KUKA KRL program: EPS_2_25252_SD6A_A_20250912064012.src

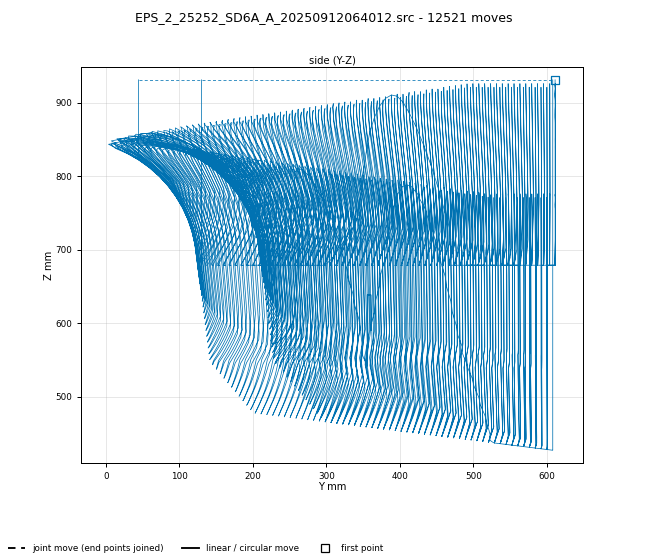
[picture p0: tool path of EPS_2_25252_SD6A_A_20250912064012.src, 12521 of 12523 moves have a stored position in this frame; points joined in program order, loops and branches not executed]
&ACCESS RVP
&REL 4
&COMMENT QRS 19112012
&PARAM EDITMASK = *
DEF PART()
EXT BAS (BAS_COMMAND :IN,REAL :IN )
INT I
BAS (#INITMOV,0 )

;KUKA QRS Post kuka4.cps  Date:22-06-2017 !

File_ID=2842

QRS_PRE_INIT()

;Init var - Until changes are made in qrs_pre_init
Outlet_Square_prg=0
Inlet_1_Square_prg=0
Inlet_2_Square_prg=0
Inlet_3_Square_prg=0
Inlet_4_Square_prg=0
Inlet_5_Square_prg=0

Outlet_1={X 0.000, Y 495.550, Z 738.000, B 0.000, E1 0.000 }
Inlet_1={X 0.000, Y 522.150, Z 645.500, B 0.000, E1 160.000 }
Outlet_1_type=366
Inlet_1_type=201
;QRS#1=Sidecore dimensions
;QRS#2=375-15" PVC SDR 35
;QRS#3=200-8" PVC SDR 35
;QRS#4=
;QRS#5=
;QRS#6=
;QRS#7=
;QRS#8=
;QRS#9=20Y PSX
;QRS#10=12-08 PSX
;QRS#11=
;QRS#12=
;QRS#13=
;QRS#14=
;QRS#15=
;QRS#16=1220x127x1219 4'
;QRS#17=EPS Height
;QRS#18=921
;QRS#19=*
;QRS#20= UPDATED VERSION 22-06-2017
;QRS#21=*
Outlet_Square=0250
Inlet_1_Square=0100
Inlet_2_Square=0
Inlet_3_Square=0
Inlet_4_Square=0
Inlet_5_Square=0
Mill_Square=1
Outlet_Square_Prg=252
Inlet_1_Square_prg=204

QRS_INIT()

$ADVANCE=5

; T1
PTP {E1 177.349,E2 177.349}
PTP {X 0,Y 611.1,A -85,B 0,C 180,E1 177.349,E2 177.349,E3 0,E4 0,E5 0,E6 0}
QRS_SPEED_INIT()
LIN {X 0,Y 611.1,Z 931,A -85,B 0,C 180,E1 177.349,E2 177.349,E3 0,E4 0,E5 0,E6 0} C_VEL
LIN {X 0,Y 611.1,Z 680.81,A -85,B 0,C 180,E1 177.349,E2 177.349} C_VEL
LIN {X 0,Y 611.172,Z 678.81,A -85,B 0,C 180,E1 177.537,E2 177.537} C_VEL
LIN {X 0,Y 611.853,Z 678.81,A -85,B 0,C 180,E1 178.833,E2 178.833} C_VEL
LIN {X 0,Y 611.873,Z 678.81,A -85,B 0,C 180,E1 185.845,E2 185.845} C_VEL
LIN {X 0,Y 611.832,Z 678.81,A -85,B 0,C 180,E1 192.946,E2 192.946} C_VEL
LIN {X 0,Y 611.828,Z 678.81,A -85,B 0,C 180,E1 200.258,E2 200.258} C_VEL
LIN {X 0,Y 611.823,Z 678.81,A -85,B 0,C 180,E1 207.934,E2 207.934} C_VEL
LIN {X 0,Y 610.481,Z 678.81,A -85,B 0,C 180,E1 210.684,E2 210.684} C_VEL
LIN {X 0,Y 611.798,Z 678.81,A -85,B 0,C 180,E1 216.206,E2 216.206} C_VEL
LIN {X 0,Y 611.214,Z 678.81,A -85,B 0,C 180,E1 217.333,E2 217.333} C_VEL
LIN {X 0,Y 610.734,Z 678.81,A -85,B 0,C 180,E1 222.325,E2 222.325} C_VEL
LIN {X 0,Y 611.755,Z 678.81,A -85,B 0,C 180,E1 224.525,E2 224.525} C_VEL
LIN {X 0,Y 611.734,Z 678.81,A -85,B 0,C 180,E1 232.604,E2 232.604} C_VEL
LIN {X 0,Y 611.207,Z 678.81,A -85,B 0,C 180,E1 233.754,E2 233.754} C_VEL
LIN {X 0,Y 611.701,Z 678.81,A -85,B 0,C 180,E1 241.161,E2 241.161} C_VEL
LIN {X 0,Y 611.507,Z 678.81,A -85,B 0,C 180,E1 242.05,E2 242.05} C_VEL
LIN {X 0,Y 611.773,Z 678.81,A -85,B 0,C 180,E1 248.631,E2 248.631} C_VEL
LIN {X 0,Y 610.949,Z 678.81,A -85,B 0,C 180,E1 248.984,E2 248.984} C_VEL
LIN {X 0,Y 610.788,Z 678.81,A -85,B 0,C 180,E1 249.001,E2 249.001} C_VEL
LIN {X 0,Y 611.596,Z 716.961,A -85,B 0,C 180,E1 249.507,E2 249.507} C_VEL
LIN {X 0,Y 611.806,Z 744.067,A -85,B 0,C 180,E1 249.858,E2 249.858} C_VEL
LIN {X 0,Y 611.827,Z 753.232,A -85,B 0,C 180,E1 250.014,E2 250.014} C_VEL
LIN {X 0,Y 611.806,Z 762.284,A -85,B 0,C 180,E1 250.207,E2 250.207} C_VEL
LIN {X 0,Y 611.661,Z 771.239,A -85,B 0,C 180,E1 250.435,E2 250.435} C_VEL
LIN {X 0,Y 611.79,Z 780.1,A -85,B 0,C 180,E1 250.71,E2 250.71} C_VEL
LIN {X 0,Y 611.791,Z 787.863,A -85,B 0,C 180,E1 250.98,E2 250.98} C_VEL
LIN {X 0,Y 611.787,Z 797.495,A -85,B 0,C 180,E1 251.365,E2 251.365} C_VEL
LIN {X 0,Y 611.804,Z 805.998,A -85,B 0,C 180,E1 251.75,E2 251.75} C_VEL
LIN {X 0,Y 611.73,Z 815.053,A -85,B 0,C 180,E1 252.208,E2 252.208} C_VEL
LIN {X 0,Y 611.709,Z 824.508,A -85,B 0,C 180,E1 252.747,E2 252.747} C_VEL
LIN {X 0,Y 611.546,Z 832.95,A -85,B 0,C 180,E1 253.278,E2 253.278} C_VEL
LIN {X 0,Y 611.448,Z 839.372,A -85,B 0,C 180,E1 253.718,E2 253.718} C_VEL
LIN {X 0,Y 611.513,Z 846.795,A -85,B 0,C 180,E1 254.279,E2 254.279} C_VEL
LIN {X 0,Y 611.729,Z 854.696,A -85,B 0,C 180,E1 254.937,E2 254.937} C_VEL
LIN {X 0,Y 611.827,Z 861.197,A -85,B 0,C 180,E1 255.523,E2 255.523} C_VEL
LIN {X 0,Y 611.641,Z 868.111,A -85,B 0,C 180,E1 256.198,E2 256.198} C_VEL
LIN {X 0,Y 611.381,Z 874.097,A -85,B 0,C 180,E1 256.831,E2 256.831} C_VEL
LIN {X 0,Y 611.254,Z 879.807,A -85,B 0,C 180,E1 257.49,E2 257.49} C_VEL
LIN {X 0,Y 611.36,Z 885.701,A -85,B 0,C 180,E1 258.239,E2 258.239} C_VEL
LIN {X 0,Y 611.556,Z 890.069,A -85,B 0,C 180,E1 258.838,E2 258.838} C_VEL
LIN {X 0,Y 611.862,Z 895.943,A -85,B 0,C 180,E1 259.735,E2 259.735} C_VEL
LIN {X 0,Y 611.484,Z 901.185,A -85,B 0,C 180,E1 260.617,E2 260.617} C_VEL
LIN {X 0,Y 611.211,Z 904.398,A -85,B 0,C 180,E1 261.204,E2 261.204} C_VEL
LIN {X 0,Y 611.059,Z 908.684,A -85,B 0,C 180,E1 262.088,E2 262.088} C_VEL
LIN {X 0,Y 611.226,Z 912.436,A -85,B 0,C 180,E1 262.974,E2 262.974} C_VEL
LIN {X 0,Y 611.629,Z 915.681,A -85,B 0,C 180,E1 263.86,E2 263.86} C_VEL
LIN {X 0,Y 611.768,Z 916.615,A -85,B 0,C 180,E1 264.154,E2 264.154} C_VEL
LIN {X 0,Y 611.736,Z 918.452,A -85,B 0,C 180,E1 264.74,E2 264.74} C_VEL
LIN {X 0,Y 611.169,Z 921.43,A -85,B 0,C 180,E1 265.908,E2 265.908} C_VEL
LIN {X 0,Y 610.976,Z 922.681,A -85,B 0,C 180,E1 266.492,E2 266.492} C_VEL
LIN {X 0,Y 611.094,Z 924.535,A -85,B 0,C 180,E1 267.712,E2 267.712} C_VEL
LIN {X 0,Y 611.599,Z 925.552,A -85,B 0,C 180,E1 268.833,E2 268.833} C_VEL
LIN {X 0,Y 611.822,Z 925.786,A -85,B 0,C 180,E1 269.3,E2 269.3} C_VEL
LIN {X 0,Y 611.469,Z 925.916,A -85,B 0,C 180,E1 270.234,E2 270.234} C_VEL
LIN {X 0,Y 611.076,Z 925.575,A -85,B 0,C 180,E1 271.168,E2 271.168} C_VEL
LIN {X 0,Y 611.003,Z 924.587,A -85,B 0,C 180,E1 272.246,E2 272.246} C_VEL
LIN {X 0,Y 611.445,Z 922.667,A -85,B 0,C 180,E1 273.505,E2 273.505} C_VEL
LIN {X 0,Y 611.74,Z 921.409,A -85,B 0,C 180,E1 274.088,E2 274.088} C_VEL
LIN {X 0,Y 611.75,Z 920.023,A -85,B 0,C 180,E1 274.674,E2 274.674} C_VEL
LIN {X 0,Y 611.456,Z 918.462,A -85,B 0,C 180,E1 275.262,E2 275.262} C_VEL
LIN {X 0,Y 611.035,Z 915.69,A -85,B 0,C 180,E1 276.146,E2 276.146} C_VEL
LIN {X 0,Y 610.903,Z 912.436,A -85,B 0,C 180,E1 277.03,E2 277.03} C_VEL
LIN {X 0,Y 611.131,Z 908.684,A -85,B 0,C 180,E1 277.911,E2 277.911} C_VEL
LIN {X 0,Y 611.584,Z 904.398,A -85,B 0,C 180,E1 278.79,E2 278.79} C_VEL
LIN {X 0,Y 611.866,Z 901.185,A -85,B 0,C 180,E1 279.377,E2 279.377} C_VEL
LIN {X 0,Y 611.515,Z 895.944,A -85,B 0,C 180,E1 280.271,E2 280.271} C_VEL
LIN {X 0,Y 611.151,Z 888.996,A -85,B 0,C 180,E1 281.318,E2 281.318} C_VEL
LIN {X 0,Y 611.162,Z 883.427,A -85,B 0,C 180,E1 282.063,E2 282.063} C_VEL
LIN {X 0,Y 611.413,Z 877.293,A -85,B 0,C 180,E1 282.806,E2 282.806} C_VEL
LIN {X 0,Y 611.786,Z 869.803,A -85,B 0,C 180,E1 283.623,E2 283.623} C_VEL
LIN {X 0,Y 611.787,Z 863.856,A -85,B 0,C 180,E1 284.223,E2 284.223} C_VEL
LIN {X 0,Y 611.564,Z 856.74,A -85,B 0,C 180,E1 284.888,E2 284.888} C_VEL
LIN {X 0,Y 611.414,Z 850.125,A -85,B 0,C 180,E1 285.456,E2 285.456} C_VEL
LIN {X 0,Y 611.435,Z 843.15,A -85,B 0,C 180,E1 286.003,E2 286.003} C_VEL
LIN {X 0,Y 611.594,Z 835.525,A -85,B 0,C 180,E1 286.548,E2 286.548} C_VEL
LIN {X 0,Y 611.771,Z 827.341,A -85,B 0,C 180,E1 287.078,E2 287.078} C_VEL
LIN {X 0,Y 611.809,Z 819.307,A -85,B 0,C 180,E1 287.555,E2 287.555} C_VEL
LIN {X 0,Y 611.791,Z 810.646,A -85,B 0,C 180,E1 288.02,E2 288.02} C_VEL
LIN {X 0,Y 611.702,Z 802.729,A -85,B 0,C 180,E1 288.407,E2 288.407} C_VEL
LIN {X 0,Y 611.705,Z 793.825,A -85,B 0,C 180,E1 288.791,E2 288.791} C_VEL
LIN {X 0,Y 611.795,Z 783.539,A -85,B 0,C 180,E1 289.174,E2 289.174} C_VEL
LIN {X 0,Y 611.762,Z 773.929,A -85,B 0,C 180,E1 289.485,E2 289.485} C_VEL
LIN {X 0,Y 611.767,Z 767.133,A -85,B 0,C 180,E1 289.678,E2 289.678} C_VEL
LIN {X 0,Y 611.841,Z 755.254,A -85,B 0,C 180,E1 289.947,E2 289.947} C_VEL
LIN {X 0,Y 611.828,Z 745.402,A -85,B 0,C 180,E1 290.122,E2 290.122} C_VEL
LIN {X 0,Y 611.684,Z 723.448,A -85,B 0,C 180,E1 290.41,E2 290.41} C_VEL
LIN {X 0,Y 610.946,Z 685.949,A -85,B 0,C 180,E1 290.897,E2 290.897} C_VEL
LIN {X 0,Y 610.763,Z 678.81,A -85,B 0,C 180,E1 290.996,E2 290.996} C_VEL
LIN {X 0,Y 611.68,Z 678.81,A -85,B 0,C 180,E1 291.148,E2 291.148} C_VEL
LIN {X 0,Y 611.713,Z 678.81,A -85,B 0,C 180,E1 291.751,E2 291.751} C_VEL
LIN {X 0,Y 611.826,Z 678.81,A -85,B 0,C 180,E1 300.61,E2 300.61} C_VEL
LIN {X 0,Y 610.649,Z 678.81,A -85,B 0,C 180,E1 307.263,E2 307.263} C_VEL
LIN {X 0,Y 611.78,Z 678.81,A -85,B 0,C 180,E1 309.156,E2 309.156} C_VEL
LIN {X 0,Y 610.375,Z 678.81,A -85,B 0,C 180,E1 312.355,E2 312.355} C_VEL
LIN {X 0,Y 610.685,Z 678.81,A -85,B 0,C 180,E1 315.577,E2 315.577} C_VEL
LIN {X 0,Y 611.769,Z 678.81,A -85,B 0,C 180,E1 317.764,E2 317.764} C_VEL
LIN {X 0,Y 610.272,Z 678.81,A -85,B 0,C 180,E1 323.689,E2 323.689} C_VEL
LIN {X 0,Y 611.793,Z 678.81,A -85,B 0,C 180,E1 326.636,E2 326.636} C_VEL
LIN {X 0,Y 611.803,Z 678.81,A -85,B 0,C 180,E1 334.676,E2 334.676} C_VEL
LIN {X 0,Y 611.537,Z 678.81,A -85,B 0,C 180,E1 343.281,E2 343.281} C_VEL
LIN {X 0,Y 611.296,Z 678.81,A -85,B 0,C 180,E1 344.633,E2 344.633} C_VEL
LIN {X 0,Y 611.872,Z 678.81,A -85,B 0,C 180,E1 351.804,E2 351.804} C_VEL
LIN {X 0,Y 611.852,Z 678.81,A -85,B 0,C 180,E1 358.833,E2 358.833} C_VEL
LIN {X 0,Y 611.874,Z 678.81,A -85,B 0,C 180,E1 368.196,E2 368.196} C_VEL
LIN {X 0,Y 611.806,Z 678.81,A -85,B 0,C 180,E1 375.354,E2 375.354} C_VEL
LIN {X 0,Y 611.825,Z 678.81,A -85,B 0,C 180,E1 382.767,E2 382.767} C_VEL
LIN {X 0,Y 611.831,Z 678.81,A -85,B 0,C 180,E1 390.609,E2 390.609} C_VEL
LIN {X 0,Y 611.757,Z 678.81,A -85,B 0,C 180,E1 399.158,E2 399.158} C_VEL
LIN {X 0,Y 610.337,Z 678.81,A -85,B 0,C 180,E1 402.359,E2 402.359} C_VEL
LIN {X 0,Y 610.636,Z 678.81,A -85,B 0,C 180,E1 405.582,E2 405.582} C_VEL
LIN {X 0,Y 611.712,Z 678.81,A -85,B 0,C 180,E1 407.759,E2 407.759} C_VEL
LIN {X 0,Y 610.218,Z 678.81,A -85,B 0,C 180,E1 413.686,E2 413.686} C_VEL
LIN {X 0,Y 611.725,Z 678.81,A -85,B 0,C 180,E1 416.637,E2 416.637} C_VEL
LIN {X 0,Y 611.755,Z 678.81,A -85,B 0,C 180,E1 424.674,E2 424.674} C_VEL
LIN {X 0,Y 611.523,Z 678.81,A -85,B 0,C 180,E1 433.285,E2 433.285} C_VEL
LIN {X 0,Y 611.29,Z 678.81,A -85,B 0,C 180,E1 434.632,E2 434.632} C_VEL
LIN {X 0,Y 611.873,Z 678.81,A -85,B 0,C 180,E1 441.804,E2 441.804} C_VEL
LIN {X 0,Y 611.873,Z 678.81,A -85,B 0,C 180,E1 448.833,E2 448.833} C_VEL
LIN {X 0,Y 611.836,Z 678.81,A -85,B 0,C 180,E1 457.976,E2 457.976} C_VEL
LIN {X 0,Y 611.68,Z 678.812,A -85,B 0,C 180,E1 458.051,E2 458.051} C_VEL
LIN {X 0,Y 611.823,Z 687.514,A -85,B 0,C 180,E1 458.307,E2 458.307} C_VEL
LIN {X 0,Y 611.725,Z 694.867,A -85,B 0,C 180,E1 458.567,E2 458.567} C_VEL
LIN {X 0,Y 611.706,Z 703.414,A -85,B 0,C 180,E1 458.936,E2 458.936} C_VEL
LIN {X 0,Y 611.787,Z 710.617,A -85,B 0,C 180,E1 459.304,E2 459.304} C_VEL
LIN {X 0,Y 611.823,Z 718.098,A -85,B 0,C 180,E1 459.747,E2 459.747} C_VEL
LIN {X 0,Y 611.74,Z 724.654,A -85,B 0,C 180,E1 460.193,E2 460.193} C_VEL
LIN {X 0,Y 611.547,Z 731.453,A -85,B 0,C 180,E1 460.716,E2 460.716} C_VEL
LIN {X 0,Y 611.554,Z 738.108,A -85,B 0,C 180,E1 461.31,E2 461.31} C_VEL
LIN {X 0,Y 611.754,Z 743.901,A -85,B 0,C 180,E1 461.902,E2 461.902} C_VEL
LIN {X 0,Y 611.846,Z 749.025,A -85,B 0,C 180,E1 462.498,E2 462.498} C_VEL
LIN {X 0,Y 611.57,Z 754.062,A -85,B 0,C 180,E1 463.155,E2 463.155} C_VEL
LIN {X 0,Y 611.352,Z 758.117,A -85,B 0,C 180,E1 463.768,E2 463.768} C_VEL
LIN {X 0,Y 611.348,Z 761.59,A -85,B 0,C 180,E1 464.365,E2 464.365} C_VEL
LIN {X 0,Y 611.521,Z 764.619,A -85,B 0,C 180,E1 464.961,E2 464.961} C_VEL
LIN {X 0,Y 611.856,Z 767.987,A -85,B 0,C 180,E1 465.746,E2 465.746} C_VEL
LIN {X 0,Y 611.76,Z 769.47,A -85,B 0,C 180,E1 466.142,E2 466.142} C_VEL
LIN {X 0,Y 611.48,Z 771.28,A -85,B 0,C 180,E1 466.702,E2 466.702} C_VEL
LIN {X 0,Y 611.285,Z 772.515,A -85,B 0,C 180,E1 467.157,E2 467.157} C_VEL
LIN {X 0,Y 611.186,Z 773.958,A -85,B 0,C 180,E1 467.808,E2 467.808} C_VEL
LIN {X 0,Y 611.315,Z 774.93,A -85,B 0,C 180,E1 468.419,E2 468.419} C_VEL
LIN {X 0,Y 611.592,Z 775.562,A -85,B 0,C 180,E1 469.026,E2 469.026} C_VEL
LIN {X 0,Y 611.86,Z 775.874,A -85,B 0,C 180,E1 469.636,E2 469.636} C_VEL
LIN {X 0,Y 611.627,Z 775.89,A -85,B 0,C 180,E1 470.265,E2 470.265} C_VEL
LIN {X 0,Y 611.328,Z 775.619,A -85,B 0,C 180,E1 470.822,E2 470.822} C_VEL
LIN {X 0,Y 611.148,Z 775.071,A -85,B 0,C 180,E1 471.378,E2 471.378} C_VEL
LIN {X 0,Y 611.15,Z 773.993,A -85,B 0,C 180,E1 472.083,E2 472.083} C_VEL
LIN {X 0,Y 611.421,Z 772.429,A -85,B 0,C 180,E1 472.783,E2 472.783} C_VEL
LIN {X 0,Y 611.84,Z 770.085,A -85,B 0,C 180,E1 473.578,E2 473.578} C_VEL
LIN {X 0,Y 611.755,Z 768.443,A -85,B 0,C 180,E1 474.044,E2 474.044} C_VEL
LIN {X 0,Y 611.36,Z 764.799,A -85,B 0,C 180,E1 474.914,E2 474.914} C_VEL
LIN {X 0,Y 611.234,Z 761.497,A -85,B 0,C 180,E1 475.563,E2 475.563} C_VEL
LIN {X 0,Y 611.357,Z 757.756,A -85,B 0,C 180,E1 476.201,E2 476.201} C_VEL
LIN {X 0,Y 611.664,Z 753.487,A -85,B 0,C 180,E1 476.834,E2 476.834} C_VEL
LIN {X 0,Y 611.854,Z 750.246,A -85,B 0,C 180,E1 477.263,E2 477.263} C_VEL
LIN {X 0,Y 611.7,Z 744.512,A -85,B 0,C 180,E1 477.94,E2 477.94} C_VEL
LIN {X 0,Y 611.466,Z 738.388,A -85,B 0,C 180,E1 478.575,E2 478.575} C_VEL
LIN {X 0,Y 611.482,Z 732.628,A -85,B 0,C 180,E1 479.094,E2 479.094} C_VEL
LIN {X 0,Y 611.679,Z 725.889,A -85,B 0,C 180,E1 479.629,E2 479.629} C_VEL
LIN {X 0,Y 611.826,Z 717.996,A -85,B 0,C 180,E1 480.169,E2 480.169} C_VEL
LIN {X 0,Y 611.747,Z 710.473,A -85,B 0,C 180,E1 480.614,E2 480.614} C_VEL
LIN {X 0,Y 611.638,Z 703.487,A -85,B 0,C 180,E1 480.972,E2 480.972} C_VEL
LIN {X 0,Y 611.645,Z 695.87,A -85,B 0,C 180,E1 481.306,E2 481.306} C_VEL
LIN {X 0,Y 611.788,Z 687.577,A -85,B 0,C 180,E1 481.601,E2 481.601} C_VEL
LIN {X 0,Y 611.726,Z 678.81,A -85,B 0,C 180,E1 481.868,E2 481.868} C_VEL
LIN {X 0,Y 611.787,Z 678.81,A -85,B 0,C 180,E1 489.156,E2 489.156} C_VEL
LIN {X 0,Y 610.358,Z 678.81,A -85,B 0,C 180,E1 492.357,E2 492.357} C_VEL
LIN {X 0,Y 610.661,Z 678.81,A -85,B 0,C 180,E1 495.58,E2 495.58} C_VEL
LIN {X 0,Y 611.745,Z 678.81,A -85,B 0,C 180,E1 497.762,E2 497.762} C_VEL
LIN {X 0,Y 611.803,Z 678.81,A -85,B 0,C 180,E1 506.626,E2 506.626} C_VEL
LIN {X 0,Y 611.822,Z 678.81,A -85,B 0,C 180,E1 514.677,E2 514.677} C_VEL
LIN {X 0,Y 611.535,Z 678.81,A -85,B 0,C 180,E1 523.281,E2 523.281} C_VEL
LIN {X 0,Y 611.283,Z 678.81,A -85,B 0,C 180,E1 524.632,E2 524.632} C_VEL
LIN {X 0,Y 611.88,Z 678.81,A -85,B 0,C 180,E1 531.804,E2 531.804} C_VEL
LIN {X 0,Y 611.172,Z 678.81,A -85,B 0,C 180,E1 537.537,E2 537.537} C_VEL
LIN {X 0,Y 602.934,Z 678.81,A -85,B 0,C 180,E1 540.812,E2 540.812} C_VEL
LIN {X 0,Y 602.904,Z 678.81,A -85,B 0,C 180,E1 547.959,E2 547.959} C_VEL
LIN {X 0,Y 602.735,Z 678.81,A -85,B 0,C 180,E1 555.332,E2 555.332} C_VEL
LIN {X 0,Y 603.135,Z 678.81,A -85,B 0,C 180,E1 561.4,E2 561.4} C_VEL
LIN {X 0,Y 602.79,Z 678.81,A -85,B 0,C 180,E1 569.709,E2 569.709} C_VEL
LIN {X 0,Y 603.079,Z 678.81,A -85,B 0,C 180,E1 577.567,E2 577.567} C_VEL
LIN {X 0,Y 602.774,Z 678.81,A -85,B 0,C 180,E1 586.184,E2 586.184} C_VEL
LIN {X 0,Y 603.193,Z 678.81,A -85,B 0,C 180,E1 593.756,E2 593.756} C_VEL
LIN {X 0,Y 603.376,Z 678.81,A -85,B 0,C 180,E1 602.271,E2 602.271} C_VEL
LIN {X 0,Y 603.322,Z 680.24,A -85,B 0,C 180,E1 608.755,E2 608.755} C_VEL
LIN {X 0,Y 604.133,Z 773.85,A -85,B 0,C 180,E1 610.257,E2 610.257} C_VEL
LIN {X 0,Y 604,Z 824.946,A -85,B 0,C 180,E1 612.547,E2 612.547} C_VEL
LIN {X 0,Y 603.791,Z 867.939,A -85,B 0,C 180,E1 615.996,E2 615.996} C_VEL
LIN {X 0,Y 603.673,Z 899.746,A -85,B 0,C 180,E1 620.23,E2 620.23} C_VEL
LIN {X 0,Y 603.606,Z 919.223,A -85,B 0,C 180,E1 624.952,E2 624.952} C_VEL
LIN {X 0,Y 603.823,Z 925.839,A -85,B 0,C 180,E1 629.28,E2 629.28} C_VEL
LIN {X 0,Y 603.745,Z 921.05,A -85,B 0,C 180,E1 634.325,E2 634.325} C_VEL
LIN {X 0,Y 603.912,Z 901.729,A -85,B 0,C 180,E1 639.401,E2 639.401} C_VEL
LIN {X 0,Y 603.891,Z 869.737,A -85,B 0,C 180,E1 643.812,E2 643.812} C_VEL
LIN {X 0,Y 604.055,Z 826.471,A -85,B 0,C 180,E1 647.357,E2 647.357} C_VEL
LIN {X 0,Y 604.212,Z 774.744,A -85,B 0,C 180,E1 649.714,E2 649.714} C_VEL
LIN {X 0,Y 603.574,Z 691.837,A -85,B 0,C 180,E1 651.091,E2 651.091} C_VEL
LIN {X 0,Y 603.706,Z 678.81,A -85,B 0,C 180,E1 651.376,E2 651.376} C_VEL
LIN {X 0,Y 603.513,Z 678.81,A -85,B 0,C 180,E1 661.029,E2 661.029} C_VEL
LIN {X 0,Y 603.293,Z 678.81,A -85,B 0,C 180,E1 669.899,E2 669.899} C_VEL
LIN {X 0,Y 603.427,Z 678.81,A -85,B 0,C 180,E1 678.202,E2 678.202} C_VEL
LIN {X 0,Y 603.246,Z 678.81,A -85,B 0,C 180,E1 687.43,E2 687.43} C_VEL
LIN {X 0,Y 603.187,Z 678.81,A -85,B 0,C 180,E1 695.47,E2 695.47} C_VEL
LIN {X 0,Y 603.261,Z 678.81,A -85,B 0,C 180,E1 704.682,E2 704.682} C_VEL
LIN {X 0,Y 602.919,Z 678.81,A -85,B 0,C 180,E1 713.833,E2 713.833} C_VEL
LIN {X 0,Y 602.552,Z 678.81,A -85,B 0,C 180,E1 720.72,E2 720.72} C_VEL
LIN {X 0,Y 603.21,Z 678.81,A -85,B 0,C 180,E1 729.411,E2 729.411} C_VEL
LIN {X 0,Y 603.008,Z 678.81,A -85,B 0,C 180,E1 736.822,E2 736.822} C_VEL
LIN {X 0,Y 602.827,Z 678.81,A -85,B 0,C 180,E1 744.542,E2 744.542} C_VEL
LIN {X 0,Y 602.654,Z 678.81,A -85,B 0,C 180,E1 752.482,E2 752.482} C_VEL
LIN {X 0,Y 603.274,Z 678.81,A -85,B 0,C 180,E1 759.901,E2 759.901} C_VEL
LIN {X 0,Y 603.368,Z 678.81,A -85,B 0,C 180,E1 768.202,E2 768.202} C_VEL
LIN {X 0,Y 603.188,Z 678.81,A -85,B 0,C 180,E1 777.441,E2 777.441} C_VEL
LIN {X 0,Y 603.142,Z 678.81,A -85,B 0,C 180,E1 785.471,E2 785.471} C_VEL
LIN {X 0,Y 603.256,Z 678.81,A -85,B 0,C 180,E1 794.684,E2 794.684} C_VEL
LIN {X 0,Y 602.922,Z 678.81,A -85,B 0,C 180,E1 803.846,E2 803.846} C_VEL
LIN {X 0,Y 602.598,Z 678.81,A -85,B 0,C 180,E1 810.722,E2 810.722} C_VEL
LIN {X 0,Y 603.887,Z 680.618,A -85,B 0,C 180,E1 817.945,E2 817.945} C_VEL
LIN {X 0,Y 603.912,Z 720.413,A -85,B 0,C 180,E1 819.766,E2 819.766} C_VEL
LIN {X 0,Y 603.781,Z 751.418,A -85,B 0,C 180,E1 822.705,E2 822.705} C_VEL
LIN {X 0,Y 603.602,Z 770.584,A -85,B 0,C 180,E1 826.43,E2 826.43} C_VEL
LIN {X 0,Y 603.782,Z 775.979,A -85,B 0,C 180,E1 829.835,E2 829.835} C_VEL
LIN {X 0,Y 603.782,Z 769.082,A -85,B 0,C 180,E1 833.931,E2 833.931} C_VEL
LIN {X 0,Y 603.788,Z 747.442,A -85,B 0,C 180,E1 837.709,E2 837.709} C_VEL
LIN {X 0,Y 603.913,Z 714.45,A -85,B 0,C 180,E1 840.524,E2 840.524} C_VEL
LIN {X 0,Y 603.549,Z 678.81,A -85,B 0,C 180,E1 842.137,E2 842.137} C_VEL
LIN {X 0,Y 603.281,Z 678.81,A -85,B 0,C 180,E1 849.9,E2 849.9} C_VEL
LIN {X 0,Y 603.388,Z 678.81,A -85,B 0,C 180,E1 858.203,E2 858.203} C_VEL
LIN {X 0,Y 603.275,Z 678.81,A -85,B 0,C 180,E1 867.426,E2 867.426} C_VEL
LIN {X 0,Y 603.228,Z 678.81,A -85,B 0,C 180,E1 875.475,E2 875.475} C_VEL
LIN {X 0,Y 603.243,Z 678.81,A -85,B 0,C 180,E1 884.685,E2 884.685} C_VEL
LIN {X 0,Y 602.93,Z 678.81,A -85,B 0,C 180,E1 893.825,E2 893.825} C_VEL
LIN {X 0,Y 602.934,Z 678.81,A -85,B 0,C 180,E1 900.812,E2 900.812} C_VEL
LIN {X 0,Y 595.014,Z 678.81,A -85,B 0,C 180,E1 904.112,E2 904.112} C_VEL
LIN {X 0,Y 595.447,Z 678.81,A -85,B 0,C 180,E1 912.513,E2 912.513} C_VEL
LIN {X 0,Y 595.014,Z 678.81,A -85,B 0,C 180,E1 921.707,E2 921.707} C_VEL
LIN {X 0,Y 594.756,Z 678.81,A -85,B 0,C 180,E1 929.842,E2 929.842} C_VEL
LIN {X 0,Y 595.449,Z 678.81,A -85,B 0,C 180,E1 936.796,E2 936.796} C_VEL
LIN {X 0,Y 595.035,Z 678.81,A -85,B 0,C 180,E1 945.465,E2 945.465} C_VEL
LIN {X 0,Y 595.252,Z 678.81,A -85,B 0,C 180,E1 953.431,E2 953.431} C_VEL
LIN {X 0,Y 595.319,Z 678.81,A -85,B 0,C 180,E1 961.862,E2 961.862} C_VEL
LIN {X 0,Y 595.753,Z 680.669,A -85,B 0,C 180,E1 968.477,E2 968.477} C_VEL
LIN {X 0,Y 596.562,Z 772.849,A -85,B 0,C 180,E1 969.966,E2 969.966} C_VEL
LIN {X 0,Y 596.266,Z 825.23,A -85,B 0,C 180,E1 972.33,E2 972.33} C_VEL
LIN {X 0,Y 595.887,Z 869.735,A -85,B 0,C 180,E1 975.999,E2 975.999} C_VEL
LIN {X 0,Y 595.563,Z 901.73,A -85,B 0,C 180,E1 980.466,E2 980.466} C_VEL
LIN {X 0,Y 595.294,Z 921.05,A -85,B 0,C 180,E1 985.614,E2 985.614} C_VEL
LIN {X 0,Y 595.235,Z 925.839,A -85,B 0,C 180,E1 990.73,E2 990.73} C_VEL
LIN {X 0,Y 595.294,Z 917.858,A -85,B 0,C 180,E1 995.615,E2 995.615} C_VEL
LIN {X 0,Y 595.497,Z 895.378,A -85,B 0,C 180,E1 1000.647,E2 1000.647} C_VEL
LIN {X 0,Y 595.923,Z 860.031,A -85,B 0,C 180,E1 1004.986,E2 1004.986} C_VEL
LIN {X 0,Y 596.451,Z 813.405,A -85,B 0,C 180,E1 1008.356,E2 1008.356} C_VEL
LIN {X 0,Y 596.771,Z 761.007,A -85,B 0,C 180,E1 1010.345,E2 1010.345} C_VEL
LIN {X 0,Y 595.496,Z 678.81,A -85,B 0,C 180,E1 1011.686,E2 1011.686} C_VEL
LIN {X 0,Y 595.195,Z 678.81,A -85,B 0,C 180,E1 1021.512,E2 1021.512} C_VEL
LIN {X 0,Y 594.689,Z 678.81,A -85,B 0,C 180,E1 1031.161,E2 1031.161} C_VEL
LIN {X 0,Y 594.698,Z 678.81,A -85,B 0,C 180,E1 1039.4,E2 1039.4} C_VEL
LIN {X 0,Y 594.769,Z 678.81,A -85,B 0,C 180,E1 1048.459,E2 1048.459} C_VEL
LIN {X 0,Y 594.527,Z 678.81,A -85,B 0,C 180,E1 1056.691,E2 1056.691} C_VEL
LIN {X 0,Y 595.268,Z 678.81,A -85,B 0,C 180,E1 1064.471,E2 1064.471} C_VEL
LIN {X 0,Y 595.065,Z 678.81,A -85,B 0,C 180,E1 1073.408,E2 1073.408} C_VEL
LIN {X 0,Y 594.542,Z 678.81,A -85,B 0,C 180,E1 1080.73,E2 1080.73} C_VEL
LIN {X 0,Y 595.149,Z 678.81,A -85,B 0,C 180,E1 1089.539,E2 1089.539} C_VEL
LIN {X 0,Y 594.912,Z 678.81,A -85,B 0,C 180,E1 1097.058,E2 1097.058} C_VEL
LIN {X 0,Y 594.658,Z 678.81,A -85,B 0,C 180,E1 1105.049,E2 1105.049} C_VEL
LIN {X 0,Y 595.183,Z 678.81,A -85,B 0,C 180,E1 1111.513,E2 1111.513} C_VEL
LIN {X 0,Y 594.663,Z 678.81,A -85,B 0,C 180,E1 1121.165,E2 1121.165} C_VEL
LIN {X 0,Y 594.646,Z 678.81,A -85,B 0,C 180,E1 1129.401,E2 1129.401} C_VEL
LIN {X 0,Y 594.697,Z 678.81,A -85,B 0,C 180,E1 1138.458,E2 1138.458} C_VEL
LIN {X 0,Y 594.465,Z 678.81,A -85,B 0,C 180,E1 1146.691,E2 1146.691} C_VEL
LIN {X 0,Y 595.261,Z 678.81,A -85,B 0,C 180,E1 1154.474,E2 1154.474} C_VEL
LIN {X 0,Y 595.076,Z 678.81,A -85,B 0,C 180,E1 1163.41,E2 1163.41} C_VEL
LIN {X 0,Y 594.588,Z 678.81,A -85,B 0,C 180,E1 1170.731,E2 1170.731} C_VEL
LIN {X 0,Y 595.818,Z 680.519,A -85,B 0,C 180,E1 1177.777,E2 1177.777} C_VEL
LIN {X 0,Y 596.015,Z 720.26,A -85,B 0,C 180,E1 1179.619,E2 1179.619} C_VEL
LIN {X 0,Y 595.814,Z 752.023,A -85,B 0,C 180,E1 1182.69,E2 1182.69} C_VEL
LIN {X 0,Y 595.5,Z 771.426,A -85,B 0,C 180,E1 1186.66,E2 1186.66} C_VEL
LIN {X 0,Y 595.63,Z 775.97,A -85,B 0,C 180,E1 1190.118,E2 1190.118} C_VEL
LIN {X 0,Y 595.655,Z 767.866,A -85,B 0,C 180,E1 1194.319,E2 1194.319} C_VEL
LIN {X 0,Y 595.762,Z 744.865,A -85,B 0,C 180,E1 1198.115,E2 1198.115} C_VEL
LIN {X 0,Y 595.979,Z 710.908,A -85,B 0,C 180,E1 1200.876,E2 1200.876} C_VEL
LIN {X 0,Y 595.427,Z 678.81,A -85,B 0,C 180,E1 1202.345,E2 1202.345} C_VEL
LIN {X 0,Y 594.679,Z 678.81,A -85,B 0,C 180,E1 1211.165,E2 1211.165} C_VEL
LIN {X 0,Y 594.648,Z 678.81,A -85,B 0,C 180,E1 1219.4,E2 1219.4} C_VEL
LIN {X 0,Y 594.781,Z 678.81,A -85,B 0,C 180,E1 1228.463,E2 1228.463} C_VEL
LIN {X 0,Y 594.516,Z 678.81,A -85,B 0,C 180,E1 1236.694,E2 1236.694} C_VEL
LIN {X 0,Y 595.249,Z 678.81,A -85,B 0,C 180,E1 1244.474,E2 1244.474} C_VEL
LIN {X 0,Y 595.068,Z 678.81,A -85,B 0,C 180,E1 1253.411,E2 1253.411} C_VEL
LIN {X 0,Y 594.952,Z 678.81,A -85,B 0,C 180,E1 1260.793,E2 1260.793} C_VEL
LIN {X 0,Y 595.014,Z 678.81,A -85,B 0,C 180,E1 1264.112,E2 1264.112} C_VEL
LIN {X 0,Y 587.07,Z 678.81,A -85,B 0,C 180,E1 1267.485,E2 1267.485} C_VEL
LIN {X 0,Y 587.131,Z 678.81,A -85,B 0,C 180,E1 1274.244,E2 1274.244} C_VEL
LIN {X 0,Y 586.879,Z 678.81,A -85,B 0,C 180,E1 1282.023,E2 1282.023} C_VEL
LIN {X 0,Y 586.599,Z 678.81,A -85,B 0,C 180,E1 1290.3,E2 1290.3} C_VEL
LIN {X 0,Y 586.867,Z 678.81,A -85,B 0,C 180,E1 1297.937,E2 1297.937} C_VEL
LIN {X 0,Y 586.568,Z 678.81,A -85,B 0,C 180,E1 1306.717,E2 1306.717} C_VEL
LIN {X 0,Y 586.75,Z 678.81,A -85,B 0,C 180,E1 1314.565,E2 1314.565} C_VEL
LIN {X 0,Y 586.929,Z 678.81,A -85,B 0,C 180,E1 1323.138,E2 1323.138} C_VEL
LIN {X 0,Y 587.554,Z 680.352,A -85,B 0,C 180,E1 1328.157,E2 1328.157} C_VEL
LIN {X 0,Y 589.018,Z 773.975,A -85,B 0,C 180,E1 1329.732,E2 1329.732} C_VEL
LIN {X 0,Y 588.575,Z 825.276,A -85,B 0,C 180,E1 1332.095,E2 1332.095} C_VEL
LIN {X 0,Y 588.038,Z 869.735,A -85,B 0,C 180,E1 1335.808,E2 1335.808} C_VEL
LIN {X 0,Y 587.653,Z 901.731,A -85,B 0,C 180,E1 1340.337,E2 1340.337} C_VEL
LIN {X 0,Y 587.323,Z 921.05,A -85,B 0,C 180,E1 1345.554,E2 1345.554} C_VEL
LIN {X 0,Y 587.23,Z 925.839,A -85,B 0,C 180,E1 1350.74,E2 1350.74} C_VEL
LIN {X 0,Y 587.257,Z 917.683,A -85,B 0,C 180,E1 1355.749,E2 1355.749} C_VEL
LIN {X 0,Y 587.519,Z 895.531,A -85,B 0,C 180,E1 1360.767,E2 1360.767} C_VEL
LIN {X 0,Y 588.045,Z 859.95,A -85,B 0,C 180,E1 1365.2,E2 1365.2} C_VEL
LIN {X 0,Y 588.78,Z 813.481,A -85,B 0,C 180,E1 1368.6,E2 1368.6} C_VEL
LIN {X 0,Y 589.251,Z 761.501,A -85,B 0,C 180,E1 1370.604,E2 1370.604} C_VEL
LIN {X 0,Y 587.286,Z 678.81,A -85,B 0,C 180,E1 1372.004,E2 1372.004} C_VEL
LIN {X 0,Y 586.895,Z 678.81,A -85,B 0,C 180,E1 1382.01,E2 1382.01} C_VEL
LIN {X 0,Y 586.652,Z 678.81,A -85,B 0,C 180,E1 1391.272,E2 1391.272} C_VEL
LIN {X 0,Y 587.074,Z 678.81,A -85,B 0,C 180,E1 1398.76,E2 1398.76} C_VEL
LIN {X 0,Y 586.839,Z 678.81,A -85,B 0,C 180,E1 1407.982,E2 1407.982} C_VEL
LIN {X 0,Y 586.543,Z 678.81,A -85,B 0,C 180,E1 1416.705,E2 1416.705} C_VEL
LIN {X 0,Y 587.247,Z 678.81,A -85,B 0,C 180,E1 1424.254,E2 1424.254} C_VEL
LIN {X 0,Y 587.088,Z 678.81,A -85,B 0,C 180,E1 1433.318,E2 1433.318} C_VEL
LIN {X 0,Y 586.528,Z 678.81,A -85,B 0,C 180,E1 1440.74,E2 1440.74} C_VEL
LIN {X 0,Y 587.118,Z 678.81,A -85,B 0,C 180,E1 1449.671,E2 1449.671} C_VEL
LIN {X 0,Y 586.83,Z 678.81,A -85,B 0,C 180,E1 1457.3,E2 1457.3} C_VEL
LIN {X 0,Y 586.605,Z 678.81,A -85,B 0,C 180,E1 1465.268,E2 1465.268} C_VEL
LIN {X 0,Y 586.537,Z 678.81,A -85,B 0,C 180,E1 1472.768,E2 1472.768} C_VEL
LIN {X 0,Y 586.624,Z 678.81,A -85,B 0,C 180,E1 1481.275,E2 1481.275} C_VEL
LIN {X 0,Y 587.019,Z 678.81,A -85,B 0,C 180,E1 1488.76,E2 1488.76} C_VEL
LIN {X 0,Y 586.767,Z 678.81,A -85,B 0,C 180,E1 1497.982,E2 1497.982} C_VEL
LIN {X 0,Y 586.443,Z 678.81,A -85,B 0,C 180,E1 1506.731,E2 1506.731} C_VEL
LIN {X 0,Y 587.238,Z 678.81,A -85,B 0,C 180,E1 1514.256,E2 1514.256} C_VEL
LIN {X 0,Y 587.099,Z 678.81,A -85,B 0,C 180,E1 1523.32,E2 1523.32} C_VEL
LIN {X 0,Y 586.575,Z 678.81,A -85,B 0,C 180,E1 1530.741,E2 1530.741} C_VEL
LIN {X 0,Y 587.52,Z 679.559,A -85,B 0,C 180,E1 1537.574,E2 1537.574} C_VEL
LIN {X 0,Y 588.142,Z 720.098,A -85,B 0,C 180,E1 1539.468,E2 1539.468} C_VEL
LIN {X 0,Y 587.929,Z 751.25,A -85,B 0,C 180,E1 1542.484,E2 1542.484} C_VEL
LIN {X 0,Y 587.585,Z 771.033,A -85,B 0,C 180,E1 1546.479,E2 1546.479} C_VEL
LIN {X 0,Y 587.514,Z 775.904,A -85,B 0,C 180,E1 1550.408,E2 1550.408} C_VEL
LIN {X 0,Y 587.62,Z 767.766,A -85,B 0,C 180,E1 1554.406,E2 1554.406} C_VEL
LIN {X 0,Y 587.823,Z 745.644,A -85,B 0,C 180,E1 1558.135,E2 1558.135} C_VEL
LIN {X 0,Y 588.118,Z 711.032,A -85,B 0,C 180,E1 1561.017,E2 1561.017} C_VEL
LIN {X 0,Y 587.385,Z 678.81,A -85,B 0,C 180,E1 1562.412,E2 1562.412} C_VEL
LIN {X 0,Y 586.64,Z 678.81,A -85,B 0,C 180,E1 1571.273,E2 1571.273} C_VEL
LIN {X 0,Y 587.029,Z 678.81,A -85,B 0,C 180,E1 1578.76,E2 1578.76} C_VEL
LIN {X 0,Y 586.844,Z 678.81,A -85,B 0,C 180,E1 1587.986,E2 1587.986} C_VEL
LIN {X 0,Y 586.501,Z 678.81,A -85,B 0,C 180,E1 1596.715,E2 1596.715} C_VEL
LIN {X 0,Y 587.229,Z 678.81,A -85,B 0,C 180,E1 1604.256,E2 1604.256} C_VEL
LIN {X 0,Y 587.091,Z 678.81,A -85,B 0,C 180,E1 1613.321,E2 1613.321} C_VEL
LIN {X 0,Y 586.964,Z 678.81,A -85,B 0,C 180,E1 1620.742,E2 1620.742} C_VEL
LIN {X 0,Y 587.07,Z 678.81,A -85,B 0,C 180,E1 1627.485,E2 1627.485} C_VEL
LIN {X 0,Y 578.875,Z 678.81,A -85,B 0,C 180,E1 1630.875,E2 1630.875} C_VEL
LIN {X 0,Y 579.097,Z 678.81,A -85,B 0,C 180,E1 1639.124,E2 1639.124} C_VEL
LIN {X 0,Y 579.049,Z 678.81,A -85,B 0,C 180,E1 1649.005,E2 1649.005} C_VEL
LIN {X 0,Y 578.846,Z 678.81,A -85,B 0,C 180,E1 1658.036,E2 1658.036} C_VEL
LIN {X 0,Y 578.748,Z 678.81,A -85,B 0,C 180,E1 1666.149,E2 1666.149} C_VEL
LIN {X 0,Y 578.836,Z 678.81,A -85,B 0,C 180,E1 1673.851,E2 1673.851} C_VEL
LIN {X 0,Y 578.981,Z 678.81,A -85,B 0,C 180,E1 1682.698,E2 1682.698} C_VEL
LIN {X 0,Y 579.345,Z 680.194,A -85,B 0,C 180,E1 1687.829,E2 1687.829} C_VEL
LIN {X 0,Y 581.543,Z 773.104,A -85,B 0,C 180,E1 1689.433,E2 1689.433} C_VEL
LIN {X 0,Y 580.905,Z 824.954,A -85,B 0,C 180,E1 1691.829,E2 1691.829} C_VEL
LIN {X 0,Y 580.265,Z 868.714,A -85,B 0,C 180,E1 1695.502,E2 1695.502} C_VEL
LIN {X 0,Y 579.713,Z 901.732,A -85,B 0,C 180,E1 1700.203,E2 1700.203} C_VEL
LIN {X 0,Y 579.371,Z 921.049,A -85,B 0,C 180,E1 1705.493,E2 1705.493} C_VEL
LIN {X 0,Y 579.239,Z 925.839,A -85,B 0,C 180,E1 1710.751,E2 1710.751} C_VEL
LIN {X 0,Y 579.222,Z 917.684,A -85,B 0,C 180,E1 1715.829,E2 1715.829} C_VEL
LIN {X 0,Y 579.51,Z 894.863,A -85,B 0,C 180,E1 1721.03,E2 1721.03} C_VEL
LIN {X 0,Y 580.165,Z 858.842,A -85,B 0,C 180,E1 1725.519,E2 1725.519} C_VEL
LIN {X 0,Y 581.14,Z 811.68,A -85,B 0,C 180,E1 1728.952,E2 1728.952} C_VEL
LIN {X 0,Y 581.83,Z 758.338,A -85,B 0,C 180,E1 1730.959,E2 1730.959} C_VEL
LIN {X 0,Y 579.146,Z 678.81,A -85,B 0,C 180,E1 1732.234,E2 1732.234} C_VEL
LIN {X 0,Y 578.656,Z 678.81,A -85,B 0,C 180,E1 1742.522,E2 1742.522} C_VEL
LIN {X 0,Y 578.554,Z 678.81,A -85,B 0,C 180,E1 1751.615,E2 1751.615} C_VEL
LIN {X 0,Y 578.442,Z 678.81,A -85,B 0,C 180,E1 1759.998,E2 1759.998} C_VEL
LIN {X 0,Y 578.66,Z 678.81,A -85,B 0,C 180,E1 1768.465,E2 1768.465} C_VEL
LIN {X 0,Y 578.713,Z 678.81,A -85,B 0,C 180,E1 1776.015,E2 1776.015} C_VEL
LIN {X 0,Y 579.208,Z 678.81,A -85,B 0,C 180,E1 1784.029,E2 1784.029} C_VEL
LIN {X 0,Y 579.107,Z 678.81,A -85,B 0,C 180,E1 1793.226,E2 1793.226} C_VEL
LIN {X 0,Y 578.514,Z 678.81,A -85,B 0,C 180,E1 1800.75,E2 1800.75} C_VEL
LIN {X 0,Y 579.063,Z 678.81,A -85,B 0,C 180,E1 1809.807,E2 1809.807} C_VEL
LIN {X 0,Y 578.782,Z 678.81,A -85,B 0,C 180,E1 1817.549,E2 1817.549} C_VEL
LIN {X 0,Y 578.526,Z 678.81,A -85,B 0,C 180,E1 1825.646,E2 1825.646} C_VEL
LIN {X 0,Y 578.635,Z 678.81,A -85,B 0,C 180,E1 1832.523,E2 1832.523} C_VEL
LIN {X 0,Y 578.523,Z 678.81,A -85,B 0,C 180,E1 1841.618,E2 1841.618} C_VEL
LIN {X 0,Y 578.393,Z 678.81,A -85,B 0,C 180,E1 1849.998,E2 1849.998} C_VEL
LIN {X 0,Y 578.591,Z 678.81,A -85,B 0,C 180,E1 1858.478,E2 1858.478} C_VEL
LIN {X 0,Y 578.666,Z 678.81,A -85,B 0,C 180,E1 1866.016,E2 1866.016} C_VEL
LIN {X 0,Y 579.196,Z 678.81,A -85,B 0,C 180,E1 1874.032,E2 1874.032} C_VEL
LIN {X 0,Y 579.118,Z 678.81,A -85,B 0,C 180,E1 1883.228,E2 1883.228} C_VEL
LIN {X 0,Y 578.562,Z 678.81,A -85,B 0,C 180,E1 1890.752,E2 1890.752} C_VEL
LIN {X 0,Y 579.547,Z 680.498,A -85,B 0,C 180,E1 1897.429,E2 1897.429} C_VEL
LIN {X 0,Y 580.227,Z 721.33,A -85,B 0,C 180,E1 1899.408,E2 1899.408} C_VEL
LIN {X 0,Y 579.943,Z 751.86,A -85,B 0,C 180,E1 1902.467,E2 1902.467} C_VEL
LIN {X 0,Y 579.578,Z 771.254,A -85,B 0,C 180,E1 1906.506,E2 1906.506} C_VEL
LIN {X 0,Y 579.426,Z 775.758,A -85,B 0,C 180,E1 1910.706,E2 1910.706} C_VEL
LIN {X 0,Y 579.405,Z 765.638,A -85,B 0,C 180,E1 1914.999,E2 1914.999} C_VEL
LIN {X 0,Y 579.705,Z 741.527,A -85,B 0,C 180,E1 1918.72,E2 1918.72} C_VEL
LIN {X 0,Y 580.201,Z 706.196,A -85,B 0,C 180,E1 1921.44,E2 1921.44} C_VEL
LIN {X 0,Y 579.257,Z 678.81,A -85,B 0,C 180,E1 1922.69,E2 1922.69} C_VEL
LIN {X 0,Y 578.538,Z 678.81,A -85,B 0,C 180,E1 1931.618,E2 1931.618} C_VEL
LIN {X 0,Y 578.385,Z 678.81,A -85,B 0,C 180,E1 1939.997,E2 1939.997} C_VEL
LIN {X 0,Y 578.671,Z 678.81,A -85,B 0,C 180,E1 1948.463,E2 1948.463} C_VEL
LIN {X 0,Y 578.718,Z 678.81,A -85,B 0,C 180,E1 1956.018,E2 1956.018} C_VEL
LIN {X 0,Y 578.762,Z 678.81,A -85,B 0,C 180,E1 1965.577,E2 1965.577} C_VEL
LIN {X 0,Y 579.111,Z 678.81,A -85,B 0,C 180,E1 1973.229,E2 1973.229} C_VEL
LIN {X 0,Y 578.984,Z 678.81,A -85,B 0,C 180,E1 1980.752,E2 1980.752} C_VEL
LIN {X 0,Y 578.836,Z 678.81,A -85,B 0,C 180,E1 1988.293,E2 1988.293} C_VEL
LIN {X 0,Y 578.875,Z 678.81,A -85,B 0,C 180,E1 1990.875,E2 1990.875} C_VEL
LIN {X 0,Y 571.047,Z 678.81,A -85,B 0,C 180,E1 1994.346,E2 1994.346} C_VEL
LIN {X 0,Y 570.686,Z 678.81,A -85,B 0,C 180,E1 2002.683,E2 2002.683} C_VEL
LIN {X 0,Y 570.62,Z 678.81,A -85,B 0,C 180,E1 2010.194,E2 2010.194} C_VEL
LIN {X 0,Y 570.635,Z 678.81,A -85,B 0,C 180,E1 2018.684,E2 2018.684} C_VEL
LIN {X 0,Y 570.401,Z 678.81,A -85,B 0,C 180,E1 2027.279,E2 2027.279} C_VEL
LIN {X 0,Y 570.47,Z 678.81,A -85,B 0,C 180,E1 2035.115,E2 2035.115} C_VEL
LIN {X 0,Y 570.726,Z 678.81,A -85,B 0,C 180,E1 2043.977,E2 2043.977} C_VEL
LIN {X 0,Y 571.264,Z 680.376,A -85,B 0,C 180,E1 2047.501,E2 2047.501} C_VEL
LIN {X 0,Y 574.223,Z 713.749,A -85,B 0,C 180,E1 2048.065,E2 2048.065} C_VEL
LIN {X 0,Y 574.017,Z 778.818,A -85,B 0,C 180,E1 2049.338,E2 2049.338} C_VEL
LIN {X 0,Y 573.115,Z 829.502,A -85,B 0,C 180,E1 2051.873,E2 2051.873} C_VEL
LIN {X 0,Y 572.211,Z 873.179,A -85,B 0,C 180,E1 2055.799,E2 2055.799} C_VEL
LIN {X 0,Y 571.624,Z 903.69,A -85,B 0,C 180,E1 2060.449,E2 2060.449} C_VEL
LIN {X 0,Y 571.393,Z 921.049,A -85,B 0,C 180,E1 2065.43,E2 2065.43} C_VEL
LIN {X 0,Y 571.235,Z 925.838,A -85,B 0,C 180,E1 2070.761,E2 2070.761} C_VEL
LIN {X 0,Y 571.154,Z 917.118,A -85,B 0,C 180,E1 2076.101,E2 2076.101} C_VEL
LIN {X 0,Y 571.516,Z 894.387,A -85,B 0,C 180,E1 2081.263,E2 2081.263} C_VEL
LIN {X 0,Y 572.327,Z 858.491,A -85,B 0,C 180,E1 2085.77,E2 2085.77} C_VEL
LIN {X 0,Y 573.491,Z 811.683,A -85,B 0,C 180,E1 2089.215,E2 2089.215} C_VEL
LIN {X 0,Y 574.367,Z 758.337,A -85,B 0,C 180,E1 2091.244,E2 2091.244} C_VEL
LIN {X 0,Y 572.085,Z 682.722,A -85,B 0,C 180,E1 2092.434,E2 2092.434} C_VEL
LIN {X 0,Y 570.898,Z 678.81,A -85,B 0,C 180,E1 2092.671,E2 2092.671} C_VEL
LIN {X 0,Y 570.96,Z 678.81,A -85,B 0,C 180,E1 2101.217,E2 2101.217} C_VEL
LIN {X 0,Y 570.715,Z 678.81,A -85,B 0,C 180,E1 2110.721,E2 2110.721} C_VEL
LIN {X 0,Y 570.658,Z 678.81,A -85,B 0,C 180,E1 2119.338,E2 2119.338} C_VEL
LIN {X 0,Y 570.596,Z 678.81,A -85,B 0,C 180,E1 2128.757,E2 2128.757} C_VEL
LIN {X 0,Y 570.496,Z 678.81,A -85,B 0,C 180,E1 2136.594,E2 2136.594} C_VEL
LIN {X 0,Y 570.832,Z 678.81,A -85,B 0,C 180,E1 2145.369,E2 2145.369} C_VEL
LIN {X 0,Y 571.121,Z 678.81,A -85,B 0,C 180,E1 2153.131,E2 2153.131} C_VEL
LIN {X 0,Y 570.502,Z 678.81,A -85,B 0,C 180,E1 2160.761,E2 2160.761} C_VEL
LIN {X 0,Y 571.037,Z 678.81,A -85,B 0,C 180,E1 2169.946,E2 2169.946} C_VEL
LIN {X 0,Y 570.719,Z 678.81,A -85,B 0,C 180,E1 2177.805,E2 2177.805} C_VEL
LIN {X 0,Y 570.47,Z 678.81,A -85,B 0,C 180,E1 2186.035,E2 2186.035} C_VEL
LIN {X 0,Y 570.441,Z 678.81,A -85,B 0,C 180,E1 2193.071,E2 2193.071} C_VEL
LIN {X 0,Y 570.686,Z 678.81,A -85,B 0,C 180,E1 2200.724,E2 2200.724} C_VEL
LIN {X 0,Y 570.609,Z 678.81,A -85,B 0,C 180,E1 2209.339,E2 2209.339} C_VEL
LIN {X 0,Y 570.537,Z 678.81,A -85,B 0,C 180,E1 2218.757,E2 2218.757} C_VEL
LIN {X 0,Y 570.417,Z 678.81,A -85,B 0,C 180,E1 2226.616,E2 2226.616} C_VEL
LIN {X 0,Y 570.831,Z 678.81,A -85,B 0,C 180,E1 2235.371,E2 2235.371} C_VEL
LIN {X 0,Y 571.132,Z 678.81,A -85,B 0,C 180,E1 2243.133,E2 2243.133} C_VEL
LIN {X 0,Y 570.549,Z 678.81,A -85,B 0,C 180,E1 2250.762,E2 2250.762} C_VEL
LIN {X 0,Y 571.421,Z 680.487,A -85,B 0,C 180,E1 2257.247,E2 2257.247} C_VEL
LIN {X 0,Y 572.343,Z 721.178,A -85,B 0,C 180,E1 2259.25,E2 2259.25} C_VEL
LIN {X 0,Y 571.947,Z 752.471,A -85,B 0,C 180,E1 2262.45,E2 2262.45} C_VEL
LIN {X 0,Y 571.704,Z 770.439,A -85,B 0,C 180,E1 2266.184,E2 2266.184} C_VEL
LIN {X 0,Y 571.412,Z 775.899,A -85,B 0,C 180,E1 2269.468,E2 2269.468} C_VEL
LIN {X 0,Y 571.746,Z 770.547,A -85,B 0,C 180,E1 2273.69,E2 2273.69} C_VEL
LIN {X 0,Y 571.94,Z 751.033,A -85,B 0,C 180,E1 2277.667,E2 2277.667} C_VEL
LIN {X 0,Y 572.347,Z 719.755,A -85,B 0,C 180,E1 2280.759,E2 2280.759} C_VEL
LIN {X 0,Y 571.2,Z 678.81,A -85,B 0,C 180,E1 2282.838,E2 2282.838} C_VEL
LIN {X 0,Y 570.711,Z 678.81,A -85,B 0,C 180,E1 2290.726,E2 2290.726} C_VEL
LIN {X 0,Y 570.615,Z 678.81,A -85,B 0,C 180,E1 2299.339,E2 2299.339} C_VEL
LIN {X 0,Y 570.605,Z 678.81,A -85,B 0,C 180,E1 2308.761,E2 2308.761} C_VEL
LIN {X 0,Y 570.468,Z 678.81,A -85,B 0,C 180,E1 2316.601,E2 2316.601} C_VEL
LIN {X 0,Y 570.819,Z 678.81,A -85,B 0,C 180,E1 2325.372,E2 2325.372} C_VEL
LIN {X 0,Y 571.125,Z 678.81,A -85,B 0,C 180,E1 2333.134,E2 2333.134} C_VEL
LIN {X 0,Y 570.979,Z 678.81,A -85,B 0,C 180,E1 2340.763,E2 2340.763} C_VEL
LIN {X 0,Y 570.816,Z 678.81,A -85,B 0,C 180,E1 2348.41,E2 2348.41} C_VEL
LIN {X 0,Y 571.047,Z 678.81,A -85,B 0,C 180,E1 2354.346,E2 2354.346} C_VEL
LIN {X 0,Y 562.706,Z 678.81,A -85,B 0,C 180,E1 2357.838,E2 2357.838} C_VEL
LIN {X 0,Y 562.807,Z 678.81,A -85,B 0,C 180,E1 2366.421,E2 2366.421} C_VEL
LIN {X 0,Y 562.868,Z 678.81,A -85,B 0,C 180,E1 2375.431,E2 2375.431} C_VEL
LIN {X 0,Y 562.712,Z 678.81,A -85,B 0,C 180,E1 2385.621,E2 2385.621} C_VEL
LIN {X 0,Y 562.594,Z 678.81,A -85,B 0,C 180,E1 2394.553,E2 2394.553} C_VEL
LIN {X 0,Y 562.779,Z 678.81,A -85,B 0,C 180,E1 2403.581,E2 2403.581} C_VEL
LIN {X 0,Y 563.178,Z 680.565,A -85,B 0,C 180,E1 2407.162,E2 2407.162} C_VEL
LIN {X 0,Y 566.568,Z 701.291,A -85,B 0,C 180,E1 2407.585,E2 2407.585} C_VEL
LIN {X 0,Y 566.5,Z 775.899,A -85,B 0,C 180,E1 2408.949,E2 2408.949} C_VEL
LIN {X 0,Y 565.474,Z 828.006,A -85,B 0,C 180,E1 2411.518,E2 2411.518} C_VEL
LIN {X 0,Y 564.487,Z 871.297,A -85,B 0,C 180,E1 2415.38,E2 2415.38} C_VEL
LIN {X 0,Y 563.698,Z 903.689,A -85,B 0,C 180,E1 2420.313,E2 2420.313} C_VEL
LIN {X 0,Y 563.343,Z 921.379,A -85,B 0,C 180,E1 2425.528,E2 2425.528} C_VEL
LIN {X 0,Y 563.23,Z 925.838,A -85,B 0,C 180,E1 2430.772,E2 2430.772} C_VEL
LIN {X 0,Y 563.141,Z 917.118,A -85,B 0,C 180,E1 2436.188,E2 2436.188} C_VEL
LIN {X 0,Y 563.571,Z 894.723,A -85,B 0,C 180,E1 2441.368,E2 2441.368} C_VEL
LIN {X 0,Y 564.503,Z 858.492,A -85,B 0,C 180,E1 2445.995,E2 2445.995} C_VEL
LIN {X 0,Y 565.865,Z 811.686,A -85,B 0,C 180,E1 2449.484,E2 2449.484} C_VEL
LIN {X 0,Y 566.916,Z 758.201,A -85,B 0,C 180,E1 2451.54,E2 2451.54} C_VEL
LIN {X 0,Y 564.457,Z 684.357,A -85,B 0,C 180,E1 2452.732,E2 2452.732} C_VEL
LIN {X 0,Y 562.735,Z 678.81,A -85,B 0,C 180,E1 2453.018,E2 2453.018} C_VEL
LIN {X 0,Y 562.755,Z 678.81,A -85,B 0,C 180,E1 2461.841,E2 2461.841} C_VEL
LIN {X 0,Y 562.533,Z 678.81,A -85,B 0,C 180,E1 2471.371,E2 2471.371} C_VEL
LIN {X 0,Y 562.731,Z 678.81,A -85,B 0,C 180,E1 2478.641,E2 2478.641} C_VEL
LIN {X 0,Y 562.618,Z 678.81,A -85,B 0,C 180,E1 2488.262,E2 2488.262} C_VEL
LIN {X 0,Y 562.363,Z 678.81,A -85,B 0,C 180,E1 2496.962,E2 2496.962} C_VEL
LIN {X 0,Y 562.857,Z 678.81,A -85,B 0,C 180,E1 2505.157,E2 2505.157} C_VEL
LIN {X 0,Y 563.131,Z 678.81,A -85,B 0,C 180,E1 2513.033,E2 2513.033} C_VEL
LIN {X 0,Y 562.515,Z 678.81,A -85,B 0,C 180,E1 2520.771,E2 2520.771} C_VEL
LIN {X 0,Y 562.939,Z 678.81,A -85,B 0,C 180,E1 2530.279,E2 2530.279} C_VEL
LIN {X 0,Y 562.669,Z 678.81,A -85,B 0,C 180,E1 2538.068,E2 2538.068} C_VEL
LIN {X 0,Y 562.588,Z 678.81,A -85,B 0,C 180,E1 2545.359,E2 2545.359} C_VEL
LIN {X 0,Y 562.314,Z 678.81,A -85,B 0,C 180,E1 2553.59,E2 2553.59} C_VEL
LIN {X 0,Y 562.358,Z 678.81,A -85,B 0,C 180,E1 2562.09,E2 2562.09} C_VEL
LIN {X 0,Y 562.305,Z 678.81,A -85,B 0,C 180,E1 2570.28,E2 2570.28} C_VEL
LIN {X 0,Y 562.557,Z 678.81,A -85,B 0,C 180,E1 2578.263,E2 2578.263} C_VEL
LIN {X 0,Y 562.304,Z 678.81,A -85,B 0,C 180,E1 2586.963,E2 2586.963} C_VEL
LIN {X 0,Y 562.854,Z 678.81,A -85,B 0,C 180,E1 2595.159,E2 2595.159} C_VEL
LIN {X 0,Y 563.141,Z 678.81,A -85,B 0,C 180,E1 2603.035,E2 2603.035} C_VEL
LIN {X 0,Y 562.562,Z 678.81,A -85,B 0,C 180,E1 2610.773,E2 2610.773} C_VEL
LIN {X 0,Y 563.288,Z 680.489,A -85,B 0,C 180,E1 2617.061,E2 2617.061} C_VEL
LIN {X 0,Y 564.443,Z 719.663,A -85,B 0,C 180,E1 2618.991,E2 2618.991} C_VEL
LIN {X 0,Y 564.011,Z 751.714,A -85,B 0,C 180,E1 2622.233,E2 2622.233} C_VEL
LIN {X 0,Y 563.609,Z 771.294,A -85,B 0,C 180,E1 2626.423,E2 2626.423} C_VEL
LIN {X 0,Y 563.403,Z 775.946,A -85,B 0,C 180,E1 2629.676,E2 2629.676} C_VEL
LIN {X 0,Y 563.701,Z 769.637,A -85,B 0,C 180,E1 2634.049,E2 2634.049} C_VEL
LIN {X 0,Y 563.971,Z 748.706,A -85,B 0,C 180,E1 2638.092,E2 2638.092} C_VEL
LIN {X 0,Y 564.489,Z 715.684,A -85,B 0,C 180,E1 2641.193,E2 2641.193} C_VEL
LIN {X 0,Y 563.115,Z 678.81,A -85,B 0,C 180,E1 2643.016,E2 2643.016} C_VEL
LIN {X 0,Y 562.378,Z 678.81,A -85,B 0,C 180,E1 2652.091,E2 2652.091} C_VEL
LIN {X 0,Y 562.296,Z 678.81,A -85,B 0,C 180,E1 2660.279,E2 2660.279} C_VEL
LIN {X 0,Y 562.621,Z 678.81,A -85,B 0,C 180,E1 2668.266,E2 2668.266} C_VEL
LIN {X 0,Y 562.344,Z 678.81,A -85,B 0,C 180,E1 2676.965,E2 2676.965} C_VEL
LIN {X 0,Y 562.842,Z 678.81,A -85,B 0,C 180,E1 2685.16,E2 2685.16} C_VEL
LIN {X 0,Y 563.135,Z 678.81,A -85,B 0,C 180,E1 2693.036,E2 2693.036} C_VEL
LIN {X 0,Y 562.98,Z 678.81,A -85,B 0,C 180,E1 2700.774,E2 2700.774} C_VEL
LIN {X 0,Y 562.795,Z 678.81,A -85,B 0,C 180,E1 2708.531,E2 2708.531} C_VEL
LIN {X 0,Y 562.603,Z 678.81,A -85,B 0,C 180,E1 2716.455,E2 2716.455} C_VEL
LIN {X 0,Y 562.706,Z 678.81,A -85,B 0,C 180,E1 2717.838,E2 2717.838} C_VEL
LIN {X 0,Y 554.911,Z 678.81,A -85,B 0,C 180,E1 2721.405,E2 2721.405} C_VEL
LIN {X 0,Y 554.582,Z 678.81,A -85,B 0,C 180,E1 2730.463,E2 2730.463} C_VEL
LIN {X 0,Y 554.541,Z 678.81,A -85,B 0,C 180,E1 2738.746,E2 2738.746} C_VEL
LIN {X 0,Y 554.544,Z 678.81,A -85,B 0,C 180,E1 2746.49,E2 2746.49} C_VEL
LIN {X 0,Y 554.626,Z 678.81,A -85,B 0,C 180,E1 2753.965,E2 2753.965} C_VEL
LIN {X 0,Y 554.784,Z 678.81,A -85,B 0,C 180,E1 2763.17,E2 2763.17} C_VEL
LIN {X 0,Y 555.05,Z 680.318,A -85,B 0,C 180,E1 2766.805,E2 2766.805} C_VEL
LIN {X 0,Y 559.145,Z 700.448,A -85,B 0,C 180,E1 2767.26,E2 2767.26} C_VEL
LIN {X 0,Y 559.004,Z 776.365,A -85,B 0,C 180,E1 2768.668,E2 2768.668} C_VEL
LIN {X 0,Y 557.836,Z 828.009,A -85,B 0,C 180,E1 2771.255,E2 2771.255} C_VEL
LIN {X 0,Y 556.659,Z 871.224,A -85,B 0,C 180,E1 2775.161,E2 2775.161} C_VEL
LIN {X 0,Y 555.761,Z 903.689,A -85,B 0,C 180,E1 2780.174,E2 2780.174} C_VEL
LIN {X 0,Y 555.452,Z 921.048,A -85,B 0,C 180,E1 2785.299,E2 2785.299} C_VEL
LIN {X 0,Y 555.226,Z 925.838,A -85,B 0,C 180,E1 2790.783,E2 2790.783} C_VEL
LIN {X 0,Y 555.135,Z 917.119,A -85,B 0,C 180,E1 2796.278,E2 2796.278} C_VEL
LIN {X 0,Y 555.628,Z 895.903,A -85,B 0,C 180,E1 2801.326,E2 2801.326} C_VEL
LIN {X 0,Y 556.696,Z 860.479,A -85,B 0,C 180,E1 2806.022,E2 2806.022} C_VEL
LIN {X 0,Y 558.206,Z 815.178,A -85,B 0,C 180,E1 2809.556,E2 2809.556} C_VEL
LIN {X 0,Y 559.378,Z 763.342,A -85,B 0,C 180,E1 2811.71,E2 2811.71} C_VEL
LIN {X 0,Y 557.13,Z 686.381,A -85,B 0,C 180,E1 2813.02,E2 2813.02} C_VEL
LIN {X 0,Y 554.561,Z 678.81,A -85,B 0,C 180,E1 2813.378,E2 2813.378} C_VEL
LIN {X 0,Y 554.622,Z 678.81,A -85,B 0,C 180,E1 2822.246,E2 2822.246} C_VEL
LIN {X 0,Y 554.543,Z 678.81,A -85,B 0,C 180,E1 2831.182,E2 2831.182} C_VEL
LIN {X 0,Y 554.399,Z 678.81,A -85,B 0,C 180,E1 2839.96,E2 2839.96} C_VEL
LIN {X 0,Y 554.646,Z 678.81,A -85,B 0,C 180,E1 2847.752,E2 2847.752} C_VEL
LIN {X 0,Y 554.418,Z 678.81,A -85,B 0,C 180,E1 2856.613,E2 2856.613} C_VEL
LIN {X 0,Y 554.867,Z 678.81,A -85,B 0,C 180,E1 2864.938,E2 2864.938} C_VEL
LIN {X 0,Y 555.143,Z 678.81,A -85,B 0,C 180,E1 2872.932,E2 2872.932} C_VEL
LIN {X 0,Y 554.502,Z 678.81,A -85,B 0,C 180,E1 2880.782,E2 2880.782} C_VEL
LIN {X 0,Y 554.964,Z 678.81,A -85,B 0,C 180,E1 2890.237,E2 2890.237} C_VEL
LIN {X 0,Y 554.627,Z 678.81,A -85,B 0,C 180,E1 2898.34,E2 2898.34} C_VEL
LIN {X 0,Y 554.436,Z 678.81,A -85,B 0,C 180,E1 2906.848,E2 2906.848} C_VEL
LIN {X 0,Y 554.19,Z 678.81,A -85,B 0,C 180,E1 2914.15,E2 2914.15} C_VEL
LIN {X 0,Y 554.364,Z 678.81,A -85,B 0,C 180,E1 2922.12,E2 2922.12} C_VEL
LIN {X 0,Y 554.355,Z 678.81,A -85,B 0,C 180,E1 2929.961,E2 2929.961} C_VEL
LIN {X 0,Y 554.586,Z 678.81,A -85,B 0,C 180,E1 2937.752,E2 2937.752} C_VEL
LIN {X 0,Y 554.36,Z 678.81,A -85,B 0,C 180,E1 2946.613,E2 2946.613} C_VEL
LIN {X 0,Y 554.862,Z 678.81,A -85,B 0,C 180,E1 2954.94,E2 2954.94} C_VEL
LIN {X 0,Y 555.152,Z 678.81,A -85,B 0,C 180,E1 2962.934,E2 2962.934} C_VEL
LIN {X 0,Y 554.55,Z 678.81,A -85,B 0,C 180,E1 2970.784,E2 2970.784} C_VEL
LIN {X 0,Y 555.152,Z 680.504,A -85,B 0,C 180,E1 2976.869,E2 2976.869} C_VEL
LIN {X 0,Y 556.576,Z 719.502,A -85,B 0,C 180,E1 2978.822,E2 2978.822} C_VEL
LIN {X 0,Y 556.072,Z 750.959,A -85,B 0,C 180,E1 2982.01,E2 2982.01} C_VEL
LIN {X 0,Y 555.755,Z 769.768,A -85,B 0,C 180,E1 2985.847,E2 2985.847} C_VEL
LIN {X 0,Y 555.371,Z 775.998,A -85,B 0,C 180,E1 2989.972,E2 2989.972} C_VEL
LIN {X 0,Y 555.637,Z 768.691,A -85,B 0,C 180,E1 2994.392,E2 2994.392} C_VEL
LIN {X 0,Y 555.983,Z 747.344,A -85,B 0,C 180,E1 2998.394,E2 2998.394} C_VEL
LIN {X 0,Y 556.62,Z 713.463,A -85,B 0,C 180,E1 3001.498,E2 3001.498} C_VEL
LIN {X 0,Y 555.011,Z 678.81,A -85,B 0,C 180,E1 3003.262,E2 3003.262} C_VEL
LIN {X 0,Y 554.383,Z 678.81,A -85,B 0,C 180,E1 3012.118,E2 3012.118} C_VEL
LIN {X 0,Y 554.35,Z 678.81,A -85,B 0,C 180,E1 3019.96,E2 3019.96} C_VEL
LIN {X 0,Y 554.641,Z 678.81,A -85,B 0,C 180,E1 3027.755,E2 3027.755} C_VEL
LIN {X 0,Y 554.404,Z 678.81,A -85,B 0,C 180,E1 3036.616,E2 3036.616} C_VEL
LIN {X 0,Y 554.851,Z 678.81,A -85,B 0,C 180,E1 3044.941,E2 3044.941} C_VEL
LIN {X 0,Y 555.147,Z 678.81,A -85,B 0,C 180,E1 3052.935,E2 3052.935} C_VEL
LIN {X 0,Y 554.975,Z 678.81,A -85,B 0,C 180,E1 3060.785,E2 3060.785} C_VEL
LIN {X 0,Y 554.802,Z 678.81,A -85,B 0,C 180,E1 3068.655,E2 3068.655} C_VEL
LIN {X 0,Y 554.604,Z 678.81,A -85,B 0,C 180,E1 3076.699,E2 3076.699} C_VEL
LIN {X 0,Y 554.911,Z 678.81,A -85,B 0,C 180,E1 3081.405,E2 3081.405} C_VEL
LIN {X 0,Y 546.516,Z 678.81,A -85,B 0,C 180,E1 3085.003,E2 3085.003} C_VEL
LIN {X 0,Y 546.4,Z 678.81,A -85,B 0,C 180,E1 3092.795,E2 3092.795} C_VEL
LIN {X 0,Y 546.439,Z 678.81,A -85,B 0,C 180,E1 3100.745,E2 3100.745} C_VEL
LIN {X 0,Y 546.399,Z 678.81,A -85,B 0,C 180,E1 3109.804,E2 3109.804} C_VEL
LIN {X 0,Y 546.509,Z 678.81,A -85,B 0,C 180,E1 3119.089,E2 3119.089} C_VEL
LIN {X 0,Y 546.89,Z 679.904,A -85,B 0,C 180,E1 3126.432,E2 3126.432} C_VEL
LIN {X 0,Y 551.819,Z 702.612,A -85,B 0,C 180,E1 3126.97,E2 3126.97} C_VEL
LIN {X 0,Y 551.56,Z 776.614,A -85,B 0,C 180,E1 3128.374,E2 3128.374} C_VEL
LIN {X 0,Y 550.2,Z 828.012,A -85,B 0,C 180,E1 3130.985,E2 3130.985} C_VEL
LIN {X 0,Y 548.854,Z 871.222,A -85,B 0,C 180,E1 3134.945,E2 3134.945} C_VEL
LIN {X 0,Y 547.86,Z 903.689,A -85,B 0,C 180,E1 3140.031,E2 3140.031} C_VEL
LIN {X 0,Y 547.472,Z 921.047,A -85,B 0,C 180,E1 3145.23,E2 3145.23} C_VEL
LIN {X 0,Y 547.23,Z 925.837,A -85,B 0,C 180,E1 3150.794,E2 3150.794} C_VEL
LIN {X 0,Y 547.246,Z 918.254,A -85,B 0,C 180,E1 3155.969,E2 3155.969} C_VEL
LIN {X 0,Y 547.683,Z 896.806,A -85,B 0,C 180,E1 3161.326,E2 3161.326} C_VEL
LIN {X 0,Y 548.866,Z 862.402,A -85,B 0,C 180,E1 3166.051,E2 3166.051} C_VEL
LIN {X 0,Y 550.567,Z 816.883,A -85,B 0,C 180,E1 3169.734,E2 3169.734} C_VEL
LIN {X 0,Y 551.934,Z 764.631,A -85,B 0,C 180,E1 3171.983,E2 3171.983} C_VEL
LIN {X 0,Y 550.049,Z 689.194,A -85,B 0,C 180,E1 3173.295,E2 3173.295} C_VEL
LIN {X 0,Y 546.425,Z 678.81,A -85,B 0,C 180,E1 3173.747,E2 3173.747} C_VEL
LIN {X 0,Y 546.482,Z 678.81,A -85,B 0,C 180,E1 3182.786,E2 3182.786} C_VEL
LIN {X 0,Y 546.569,Z 678.81,A -85,B 0,C 180,E1 3190.729,E2 3190.729} C_VEL
LIN {X 0,Y 546.434,Z 678.81,A -85,B 0,C 180,E1 3199.794,E2 3199.794} C_VEL
LIN {X 0,Y 546.447,Z 678.81,A -85,B 0,C 180,E1 3209.081,E2 3209.081} C_VEL
LIN {X 0,Y 546.51,Z 678.81,A -85,B 0,C 180,E1 3216.254,E2 3216.254} C_VEL
LIN {X 0,Y 546.869,Z 678.81,A -85,B 0,C 180,E1 3224.712,E2 3224.712} C_VEL
LIN {X 0,Y 547.144,Z 678.81,A -85,B 0,C 180,E1 3232.828,E2 3232.828} C_VEL
LIN {X 0,Y 546.501,Z 678.81,A -85,B 0,C 180,E1 3240.794,E2 3240.794} C_VEL
LIN {X 0,Y 546.918,Z 678.81,A -85,B 0,C 180,E1 3250.389,E2 3250.389} C_VEL
LIN {X 0,Y 546.625,Z 678.81,A -85,B 0,C 180,E1 3258.618,E2 3258.618} C_VEL
LIN {X 0,Y 546.493,Z 678.81,A -85,B 0,C 180,E1 3267.27,E2 3267.27} C_VEL
LIN {X 0,Y 546.135,Z 678.81,A -85,B 0,C 180,E1 3274.944,E2 3274.944} C_VEL
LIN {X 0,Y 546.272,Z 678.81,A -85,B 0,C 180,E1 3282.892,E2 3282.892} C_VEL
LIN {X 0,Y 546.391,Z 678.81,A -85,B 0,C 180,E1 3289.8,E2 3289.8} C_VEL
LIN {X 0,Y 546.355,Z 678.81,A -85,B 0,C 180,E1 3299.079,E2 3299.079} C_VEL
LIN {X 0,Y 546.456,Z 678.81,A -85,B 0,C 180,E1 3306.255,E2 3306.255} C_VEL
LIN {X 0,Y 546.864,Z 678.81,A -85,B 0,C 180,E1 3314.715,E2 3314.715} C_VEL
LIN {X 0,Y 547.153,Z 678.81,A -85,B 0,C 180,E1 3322.83,E2 3322.83} C_VEL
LIN {X 0,Y 546.547,Z 678.81,A -85,B 0,C 180,E1 3330.796,E2 3330.796} C_VEL
LIN {X 0,Y 547.06,Z 680.473,A -85,B 0,C 180,E1 3336.671,E2 3336.671} C_VEL
LIN {X 0,Y 548.707,Z 716.567,A -85,B 0,C 180,E1 3338.449,E2 3338.449} C_VEL
LIN {X 0,Y 548.103,Z 748.739,A -85,B 0,C 180,E1 3341.585,E2 3341.585} C_VEL
LIN {X 0,Y 547.773,Z 769.417,A -85,B 0,C 180,E1 3345.671,E2 3345.671} C_VEL
LIN {X 0,Y 547.33,Z 775.937,A -85,B 0,C 180,E1 3350.278,E2 3350.278} C_VEL
LIN {X 0,Y 547.52,Z 767.474,A -85,B 0,C 180,E1 3354.816,E2 3354.816} C_VEL
LIN {X 0,Y 547.958,Z 744.664,A -85,B 0,C 180,E1 3358.857,E2 3358.857} C_VEL
LIN {X 0,Y 548.74,Z 709.536,A -85,B 0,C 180,E1 3361.912,E2 3361.912} C_VEL
LIN {X 0,Y 546.945,Z 678.81,A -85,B 0,C 180,E1 3363.408,E2 3363.408} C_VEL
LIN {X 0,Y 546.309,Z 678.81,A -85,B 0,C 180,E1 3372.888,E2 3372.888} C_VEL
LIN {X 0,Y 546.388,Z 678.81,A -85,B 0,C 180,E1 3379.799,E2 3379.799} C_VEL
LIN {X 0,Y 546.45,Z 678.81,A -85,B 0,C 180,E1 3389.085,E2 3389.085} C_VEL
LIN {X 0,Y 546.5,Z 678.81,A -85,B 0,C 180,E1 3396.257,E2 3396.257} C_VEL
LIN {X 0,Y 546.853,Z 678.81,A -85,B 0,C 180,E1 3404.715,E2 3404.715} C_VEL
LIN {X 0,Y 547.148,Z 678.81,A -85,B 0,C 180,E1 3412.831,E2 3412.831} C_VEL
LIN {X 0,Y 546.985,Z 678.81,A -85,B 0,C 180,E1 3420.796,E2 3420.796} C_VEL
LIN {X 0,Y 546.786,Z 678.81,A -85,B 0,C 180,E1 3428.782,E2 3428.782} C_VEL
LIN {X 0,Y 546.631,Z 678.81,A -85,B 0,C 180,E1 3436.95,E2 3436.95} C_VEL
LIN {X 0,Y 546.516,Z 678.81,A -85,B 0,C 180,E1 3445.003,E2 3445.003} C_VEL
LIN {X 0,Y 538.674,Z 678.81,A -85,B 0,C 180,E1 3448.673,E2 3448.673} C_VEL
LIN {X 0,Y 538.691,Z 678.81,A -85,B 0,C 180,E1 3457.282,E2 3457.282} C_VEL
LIN {X 0,Y 538.463,Z 678.81,A -85,B 0,C 180,E1 3466.332,E2 3466.332} C_VEL
LIN {X 0,Y 538.394,Z 678.81,A -85,B 0,C 180,E1 3474.702,E2 3474.702} C_VEL
LIN {X 0,Y 538.674,Z 678.81,A -85,B 0,C 180,E1 3484.109,E2 3484.109} C_VEL
LIN {X 0,Y 538.868,Z 680.112,A -85,B 0,C 180,E1 3486.08,E2 3486.08} C_VEL
LIN {X 0,Y 544.467,Z 702.491,A -85,B 0,C 180,E1 3486.639,E2 3486.639} C_VEL
LIN {X 0,Y 544.142,Z 776.04,A -85,B 0,C 180,E1 3488.044,E2 3488.044} C_VEL
LIN {X 0,Y 542.552,Z 828.014,A -85,B 0,C 180,E1 3490.707,E2 3490.707} C_VEL
LIN {X 0,Y 541.038,Z 871.058,A -85,B 0,C 180,E1 3494.703,E2 3494.703} C_VEL
LIN {X 0,Y 539.933,Z 903.688,A -85,B 0,C 180,E1 3499.883,E2 3499.883} C_VEL
LIN {X 0,Y 539.509,Z 921.047,A -85,B 0,C 180,E1 3505.159,E2 3505.159} C_VEL
LIN {X 0,Y 539.226,Z 925.837,A -85,B 0,C 180,E1 3510.806,E2 3510.806} C_VEL
LIN {X 0,Y 539.227,Z 918.254,A -85,B 0,C 180,E1 3516.058,E2 3516.058} C_VEL
LIN {X 0,Y 539.687,Z 896.479,A -85,B 0,C 180,E1 3521.557,E2 3521.557} C_VEL
LIN {X 0,Y 541.029,Z 862.401,A -85,B 0,C 180,E1 3526.29,E2 3526.29} C_VEL
LIN {X 0,Y 542.942,Z 816.88,A -85,B 0,C 180,E1 3530.023,E2 3530.023} C_VEL
LIN {X 0,Y 544.522,Z 764.63,A -85,B 0,C 180,E1 3532.298,E2 3532.298} C_VEL
LIN {X 0,Y 542.426,Z 690.257,A -85,B 0,C 180,E1 3533.627,E2 3533.627} C_VEL
LIN {X 0,Y 538.296,Z 678.81,A -85,B 0,C 180,E1 3534.128,E2 3534.128} C_VEL
LIN {X 0,Y 538.324,Z 678.81,A -85,B 0,C 180,E1 3543.347,E2 3543.347} C_VEL
LIN {X 0,Y 538.387,Z 678.81,A -85,B 0,C 180,E1 3551.667,E2 3551.667} C_VEL
LIN {X 0,Y 538.222,Z 678.81,A -85,B 0,C 180,E1 3560.839,E2 3560.839} C_VEL
LIN {X 0,Y 538.41,Z 678.81,A -85,B 0,C 180,E1 3569.279,E2 3569.279} C_VEL
LIN {X 0,Y 538.171,Z 678.81,A -85,B 0,C 180,E1 3577.621,E2 3577.621} C_VEL
LIN {X 0,Y 538.59,Z 678.81,A -85,B 0,C 180,E1 3586.141,E2 3586.141} C_VEL
LIN {X 0,Y 538.887,Z 678.81,A -85,B 0,C 180,E1 3594.342,E2 3594.342} C_VEL
LIN {X 0,Y 538.507,Z 678.81,A -85,B 0,C 180,E1 3600.806,E2 3600.806} C_VEL
LIN {X 0,Y 538.876,Z 678.81,A -85,B 0,C 180,E1 3610.546,E2 3610.546} C_VEL
LIN {X 0,Y 538.584,Z 678.81,A -85,B 0,C 180,E1 3619.28,E2 3619.28} C_VEL
LIN {X 0,Y 538.492,Z 678.81,A -85,B 0,C 180,E1 3627.71,E2 3627.71} C_VEL
LIN {X 0,Y 538.209,Z 678.81,A -85,B 0,C 180,E1 3636.526,E2 3636.526} C_VEL
LIN {X 0,Y 538.523,Z 678.81,A -85,B 0,C 180,E1 3646.338,E2 3646.338} C_VEL
LIN {X 0,Y 538.504,Z 678.81,A -85,B 0,C 180,E1 3656.666,E2 3656.666} C_VEL
LIN {X 0,Y 538.424,Z 678.81,A -85,B 0,C 180,E1 3666.353,E2 3666.353} C_VEL
LIN {X 0,Y 538.859,Z 678.81,A -85,B 0,C 180,E1 3674.482,E2 3674.482} C_VEL
LIN {X 0,Y 539.149,Z 678.81,A -85,B 0,C 180,E1 3682.723,E2 3682.723} C_VEL
LIN {X 0,Y 538.538,Z 678.81,A -85,B 0,C 180,E1 3690.807,E2 3690.807} C_VEL
LIN {X 0,Y 538.907,Z 680.376,A -85,B 0,C 180,E1 3696.463,E2 3696.463} C_VEL
LIN {X 0,Y 540.918,Z 713.332,A -85,B 0,C 180,E1 3698.064,E2 3698.064} C_VEL
LIN {X 0,Y 540.101,Z 746.365,A -85,B 0,C 180,E1 3701.138,E2 3701.138} C_VEL
LIN {X 0,Y 539.682,Z 767.685,A -85,B 0,C 180,E1 3705.084,E2 3705.084} C_VEL
LIN {X 0,Y 539.299,Z 775.909,A -85,B 0,C 180,E1 3709.492,E2 3709.492} C_VEL
LIN {X 0,Y 539.695,Z 770.122,A -85,B 0,C 180,E1 3714.062,E2 3714.062} C_VEL
LIN {X 0,Y 540.075,Z 749.598,A -85,B 0,C 180,E1 3718.331,E2 3718.331} C_VEL
LIN {X 0,Y 540.871,Z 717.119,A -85,B 0,C 180,E1 3721.59,E2 3721.59} C_VEL
LIN {X 0,Y 539.305,Z 681.198,A -85,B 0,C 180,E1 3723.411,E2 3723.411} C_VEL
LIN {X 0,Y 538.839,Z 678.81,A -85,B 0,C 180,E1 3723.816,E2 3723.816} C_VEL
LIN {X 0,Y 538.393,Z 678.81,A -85,B 0,C 180,E1 3731.673,E2 3731.673} C_VEL
LIN {X 0,Y 538.148,Z 678.81,A -85,B 0,C 180,E1 3740.849,E2 3740.849} C_VEL
LIN {X 0,Y 538.417,Z 678.81,A -85,B 0,C 180,E1 3749.278,E2 3749.278} C_VEL
LIN {X 0,Y 538.161,Z 678.81,A -85,B 0,C 180,E1 3757.625,E2 3757.625} C_VEL
LIN {X 0,Y 538.562,Z 678.81,A -85,B 0,C 180,E1 3766.442,E2 3766.442} C_VEL
LIN {X 0,Y 538.895,Z 678.81,A -85,B 0,C 180,E1 3774.345,E2 3774.345} C_VEL
LIN {X 0,Y 538.876,Z 678.81,A -85,B 0,C 180,E1 3781.335,E2 3781.335} C_VEL
LIN {X 0,Y 538.788,Z 678.81,A -85,B 0,C 180,E1 3788.914,E2 3788.914} C_VEL
LIN {X 0,Y 538.632,Z 678.81,A -85,B 0,C 180,E1 3797.21,E2 3797.21} C_VEL
LIN {X 0,Y 538.623,Z 678.81,A -85,B 0,C 180,E1 3805.897,E2 3805.897} C_VEL
LIN {X 0,Y 538.674,Z 678.81,A -85,B 0,C 180,E1 3808.673,E2 3808.673} C_VEL
LIN {X 0,Y 530.343,Z 678.81,A -85,B 0,C 180,E1 3812.361,E2 3812.361} C_VEL
LIN {X 0,Y 530.382,Z 678.81,A -85,B 0,C 180,E1 3820.692,E2 3820.692} C_VEL
LIN {X 0,Y 530.327,Z 678.81,A -85,B 0,C 180,E1 3829.921,E2 3829.921} C_VEL
LIN {X 0,Y 530.286,Z 678.81,A -85,B 0,C 180,E1 3838.033,E2 3838.033} C_VEL
LIN {X 0,Y 530.759,Z 679.764,A -85,B 0,C 180,E1 3845.779,E2 3845.779} C_VEL
LIN {X 0,Y 537.039,Z 702.919,A -85,B 0,C 180,E1 3846.328,E2 3846.328} C_VEL
LIN {X 0,Y 536.708,Z 776.059,A -85,B 0,C 180,E1 3847.724,E2 3847.724} C_VEL
LIN {X 0,Y 534.916,Z 828.017,A -85,B 0,C 180,E1 3850.42,E2 3850.42} C_VEL
LIN {X 0,Y 533.24,Z 870.858,A -85,B 0,C 180,E1 3854.45,E2 3854.45} C_VEL
LIN {X 0,Y 532.026,Z 903.469,A -85,B 0,C 180,E1 3859.684,E2 3859.684} C_VEL
LIN {X 0,Y 531.535,Z 921.046,A -85,B 0,C 180,E1 3865.086,E2 3865.086} C_VEL
LIN {X 0,Y 531.239,Z 925.837,A -85,B 0,C 180,E1 3870.818,E2 3870.818} C_VEL
LIN {X 0,Y 531.222,Z 918.254,A -85,B 0,C 180,E1 3876.15,E2 3876.15} C_VEL
LIN {X 0,Y 531.75,Z 897.568,A -85,B 0,C 180,E1 3881.523,E2 3881.523} C_VEL
LIN {X 0,Y 533.218,Z 864.323,A -85,B 0,C 180,E1 3886.322,E2 3886.322} C_VEL
LIN {X 0,Y 535.318,Z 818.727,A -85,B 0,C 180,E1 3890.203,E2 3890.203} C_VEL
LIN {X 0,Y 537.05,Z 766.743,A -85,B 0,C 180,E1 3892.567,E2 3892.567} C_VEL
LIN {X 0,Y 535.08,Z 692.707,A -85,B 0,C 180,E1 3893.885,E2 3893.885} C_VEL
LIN {X 0,Y 530.233,Z 678.81,A -85,B 0,C 180,E1 3894.38,E2 3894.38} C_VEL
LIN {X 0,Y 530.422,Z 678.81,A -85,B 0,C 180,E1 3902.427,E2 3902.427} C_VEL
LIN {X 0,Y 530.29,Z 678.81,A -85,B 0,C 180,E1 3912.261,E2 3912.261} C_VEL
LIN {X 0,Y 530.28,Z 678.81,A -85,B 0,C 180,E1 3919.912,E2 3919.912} C_VEL
LIN {X 0,Y 530.459,Z 678.81,A -85,B 0,C 180,E1 3928.041,E2 3928.041} C_VEL
LIN {X 0,Y 530.233,Z 678.81,A -85,B 0,C 180,E1 3937.268,E2 3937.268} C_VEL
LIN {X 0,Y 530.601,Z 678.81,A -85,B 0,C 180,E1 3945.928,E2 3945.928} C_VEL
LIN {X 0,Y 530.891,Z 678.81,A -85,B 0,C 180,E1 3954.256,E2 3954.256} C_VEL
LIN {X 0,Y 530.494,Z 678.81,A -85,B 0,C 180,E1 3960.818,E2 3960.818} C_VEL
LIN {X 0,Y 530.855,Z 678.81,A -85,B 0,C 180,E1 3970.708,E2 3970.708} C_VEL
LIN {X 0,Y 530.598,Z 678.81,A -85,B 0,C 180,E1 3979.202,E2 3979.202} C_VEL
LIN {X 0,Y 530.482,Z 678.81,A -85,B 0,C 180,E1 3988.165,E2 3988.165} C_VEL
LIN {X 0,Y 530.343,Z 678.81,A -85,B 0,C 180,E1 3998.104,E2 3998.104} C_VEL
LIN {X 0,Y 530.486,Z 678.81,A -85,B 0,C 180,E1 4007.759,E2 4007.759} C_VEL
LIN {X 0,Y 530.389,Z 678.81,A -85,B 0,C 180,E1 4018.04,E2 4018.04} C_VEL
LIN {X 0,Y 530.163,Z 678.81,A -85,B 0,C 180,E1 4027.268,E2 4027.268} C_VEL
LIN {X 0,Y 530.605,Z 678.81,A -85,B 0,C 180,E1 4035.93,E2 4035.93} C_VEL
LIN {X 0,Y 530.904,Z 678.81,A -85,B 0,C 180,E1 4044.258,E2 4044.258} C_VEL
LIN {X 0,Y 530.526,Z 678.81,A -85,B 0,C 180,E1 4050.82,E2 4050.82} C_VEL
LIN {X 0,Y 530.706,Z 679.913,A -85,B 0,C 180,E1 4056.156,E2 4056.156} C_VEL
LIN {X 0,Y 533.231,Z 708.781,A -85,B 0,C 180,E1 4057.564,E2 4057.564} C_VEL
LIN {X 0,Y 532.137,Z 743.862,A -85,B 0,C 180,E1 4060.683,E2 4060.683} C_VEL
LIN {X 0,Y 531.652,Z 767.244,A -85,B 0,C 180,E1 4064.886,E2 4064.886} C_VEL
LIN {X 0,Y 531.298,Z 775.784,A -85,B 0,C 180,E1 4069.176,E2 4069.176} C_VEL
LIN {X 0,Y 531.701,Z 770.605,A -85,B 0,C 180,E1 4073.951,E2 4073.951} C_VEL
LIN {X 0,Y 532.138,Z 751.432,A -85,B 0,C 180,E1 4078.187,E2 4078.187} C_VEL
LIN {X 0,Y 533.035,Z 719.154,A -85,B 0,C 180,E1 4081.641,E2 4081.641} C_VEL
LIN {X 0,Y 531.669,Z 682.731,A -85,B 0,C 180,E1 4083.637,E2 4083.637} C_VEL
LIN {X 0,Y 530.821,Z 678.81,A -85,B 0,C 180,E1 4083.882,E2 4083.882} C_VEL
LIN {X 0,Y 530.254,Z 678.81,A -85,B 0,C 180,E1 4093.13,E2 4093.13} C_VEL
LIN {X 0,Y 530.016,Z 678.81,A -85,B 0,C 180,E1 4102.005,E2 4102.005} C_VEL
LIN {X 0,Y 530.367,Z 678.81,A -85,B 0,C 180,E1 4110.774,E2 4110.774} C_VEL
LIN {X 0,Y 530.021,Z 678.81,A -85,B 0,C 180,E1 4119.029,E2 4119.029} C_VEL
LIN {X 0,Y 530.598,Z 678.81,A -85,B 0,C 180,E1 4125.931,E2 4125.931} C_VEL
LIN {X 0,Y 530.898,Z 678.81,A -85,B 0,C 180,E1 4134.26,E2 4134.26} C_VEL
LIN {X 0,Y 531.002,Z 678.81,A -85,B 0,C 180,E1 4140.82,E2 4140.82} C_VEL
LIN {X 0,Y 530.745,Z 678.81,A -85,B 0,C 180,E1 4149.442,E2 4149.442} C_VEL
LIN {X 0,Y 530.64,Z 678.81,A -85,B 0,C 180,E1 4157.477,E2 4157.477} C_VEL
LIN {X 0,Y 530.65,Z 678.81,A -85,B 0,C 180,E1 4166.316,E2 4166.316} C_VEL
LIN {X 0,Y 530.343,Z 678.81,A -85,B 0,C 180,E1 4172.361,E2 4172.361} C_VEL
LIN {X 0,Y 522.484,Z 678.81,A -85,B 0,C 180,E1 4176.138,E2 4176.138} C_VEL
LIN {X 0,Y 522.499,Z 678.81,A -85,B 0,C 180,E1 4185.369,E2 4185.369} C_VEL
LIN {X 0,Y 522.283,Z 678.81,A -85,B 0,C 180,E1 4195.487,E2 4195.487} C_VEL
LIN {X 0,Y 522.638,Z 678.81,A -85,B 0,C 180,E1 4205.101,E2 4205.101} C_VEL
LIN {X 0,Y 523.234,Z 681.76,A -85,B 0,C 180,E1 4205.526,E2 4205.526} C_VEL
LIN {X 0,Y 529.497,Z 705.834,A -85,B 0,C 180,E1 4206.096,E2 4206.096} C_VEL
LIN {X 0,Y 529.085,Z 777.292,A -85,B 0,C 180,E1 4207.497,E2 4207.497} C_VEL
LIN {X 0,Y 527.291,Z 828.605,A -85,B 0,C 180,E1 4210.168,E2 4210.168} C_VEL
LIN {X 0,Y 525.392,Z 871.491,A -85,B 0,C 180,E1 4214.289,E2 4214.289} C_VEL
LIN {X 0,Y 524.129,Z 902.991,A -85,B 0,C 180,E1 4219.424,E2 4219.424} C_VEL
LIN {X 0,Y 523.578,Z 921.046,A -85,B 0,C 180,E1 4225.012,E2 4225.012} C_VEL
LIN {X 0,Y 523.252,Z 925.837,A -85,B 0,C 180,E1 4230.831,E2 4230.831} C_VEL
LIN {X 0,Y 523.238,Z 918.254,A -85,B 0,C 180,E1 4236.244,E2 4236.244} C_VEL
LIN {X 0,Y 523.786,Z 897.568,A -85,B 0,C 180,E1 4241.701,E2 4241.701} C_VEL
LIN {X 0,Y 525.372,Z 864.322,A -85,B 0,C 180,E1 4246.573,E2 4246.573} C_VEL
LIN {X 0,Y 527.708,Z 819.277,A -85,B 0,C 180,E1 4250.469,E2 4250.469} C_VEL
LIN {X 0,Y 529.481,Z 766.883,A -85,B 0,C 180,E1 4252.835,E2 4252.835} C_VEL
LIN {X 0,Y 527.473,Z 694.523,A -85,B 0,C 180,E1 4254.143,E2 4254.143} C_VEL
LIN {X 0,Y 522.163,Z 678.81,A -85,B 0,C 180,E1 4254.729,E2 4254.729} C_VEL
LIN {X 0,Y 522.226,Z 678.81,A -85,B 0,C 180,E1 4264.079,E2 4264.079} C_VEL
LIN {X 0,Y 522.267,Z 678.81,A -85,B 0,C 180,E1 4273.066,E2 4273.066} C_VEL
LIN {X 0,Y 522.091,Z 678.81,A -85,B 0,C 180,E1 4281.318,E2 4281.318} C_VEL
LIN {X 0,Y 522.322,Z 678.81,A -85,B 0,C 180,E1 4289.436,E2 4289.436} C_VEL
LIN {X 0,Y 522.256,Z 678.81,A -85,B 0,C 180,E1 4296.901,E2 4296.901} C_VEL
LIN {X 0,Y 522.619,Z 678.81,A -85,B 0,C 180,E1 4305.708,E2 4305.708} C_VEL
LIN {X 0,Y 522.909,Z 678.81,A -85,B 0,C 180,E1 4314.168,E2 4314.168} C_VEL
LIN {X 0,Y 522.481,Z 678.81,A -85,B 0,C 180,E1 4320.83,E2 4320.83} C_VEL
LIN {X 0,Y 523.183,Z 678.81,A -85,B 0,C 180,E1 4329.179,E2 4329.179} C_VEL
LIN {X 0,Y 522.763,Z 678.81,A -85,B 0,C 180,E1 4337.746,E2 4337.746} C_VEL
LIN {X 0,Y 522.463,Z 678.81,A -85,B 0,C 180,E1 4346.757,E2 4346.757} C_VEL
LIN {X 0,Y 522.165,Z 678.81,A -85,B 0,C 180,E1 4354.522,E2 4354.522} C_VEL
LIN {X 0,Y 522.22,Z 678.81,A -85,B 0,C 180,E1 4363.071,E2 4363.071} C_VEL
LIN {X 0,Y 522.042,Z 678.81,A -85,B 0,C 180,E1 4371.318,E2 4371.318} C_VEL
LIN {X 0,Y 522.251,Z 678.81,A -85,B 0,C 180,E1 4379.435,E2 4379.435} C_VEL
LIN {X 0,Y 522.19,Z 678.81,A -85,B 0,C 180,E1 4386.901,E2 4386.901} C_VEL
LIN {X 0,Y 522.622,Z 678.81,A -85,B 0,C 180,E1 4395.711,E2 4395.711} C_VEL
LIN {X 0,Y 522.922,Z 678.81,A -85,B 0,C 180,E1 4404.17,E2 4404.17} C_VEL
LIN {X 0,Y 522.513,Z 678.81,A -85,B 0,C 180,E1 4410.832,E2 4410.832} C_VEL
LIN {X 0,Y 522.747,Z 680.74,A -85,B 0,C 180,E1 4415.884,E2 4415.884} C_VEL
LIN {X 0,Y 525.642,Z 708.414,A -85,B 0,C 180,E1 4417.256,E2 4417.256} C_VEL
LIN {X 0,Y 524.395,Z 742.988,A -85,B 0,C 180,E1 4420.295,E2 4420.295} C_VEL
LIN {X 0,Y 523.616,Z 765.69,A -85,B 0,C 180,E1 4424.262,E2 4424.262} C_VEL
LIN {X 0,Y 523.371,Z 774.573,A -85,B 0,C 180,E1 4427.725,E2 4427.725} C_VEL
LIN {X 0,Y 523.401,Z 774.572,A -85,B 0,C 180,E1 4432.189,E2 4432.189} C_VEL
LIN {X 0,Y 523.758,Z 761.301,A -85,B 0,C 180,E1 4436.686,E2 4436.686} C_VEL
LIN {X 0,Y 524.719,Z 734.863,A -85,B 0,C 180,E1 4440.551,E2 4440.551} C_VEL
LIN {X 0,Y 525.944,Z 697.665,A -85,B 0,C 180,E1 4443.251,E2 4443.251} C_VEL
LIN {X 0,Y 522.757,Z 678.81,A -85,B 0,C 180,E1 4444.171,E2 4444.171} C_VEL
LIN {X 0,Y 522.255,Z 678.81,A -85,B 0,C 180,E1 4453.067,E2 4453.067} C_VEL
LIN {X 0,Y 522.031,Z 678.81,A -85,B 0,C 180,E1 4461.317,E2 4461.317} C_VEL
LIN {X 0,Y 522.329,Z 678.81,A -85,B 0,C 180,E1 4469.44,E2 4469.44} C_VEL
LIN {X 0,Y 522.248,Z 678.81,A -85,B 0,C 180,E1 4476.904,E2 4476.904} C_VEL
LIN {X 0,Y 522.614,Z 678.81,A -85,B 0,C 180,E1 4485.712,E2 4485.712} C_VEL
LIN {X 0,Y 522.916,Z 678.81,A -85,B 0,C 180,E1 4494.172,E2 4494.172} C_VEL
LIN {X 0,Y 523.008,Z 678.81,A -85,B 0,C 180,E1 4500.833,E2 4500.833} C_VEL
LIN {X 0,Y 522.769,Z 678.81,A -85,B 0,C 180,E1 4509.189,E2 4509.189} C_VEL
LIN {X 0,Y 522.644,Z 678.81,A -85,B 0,C 180,E1 4517.754,E2 4517.754} C_VEL
LIN {X 0,Y 522.658,Z 678.81,A -85,B 0,C 180,E1 4527.678,E2 4527.678} C_VEL
LIN {X 0,Y 522.484,Z 678.81,A -85,B 0,C 180,E1 4536.138,E2 4536.138} C_VEL
LIN {X 0,Y 514.319,Z 678.81,A -85,B 0,C 180,E1 4539.973,E2 4539.973} C_VEL
LIN {X 0,Y 514.262,Z 678.81,A -85,B 0,C 180,E1 4548.812,E2 4548.812} C_VEL
LIN {X 0,Y 514.228,Z 678.81,A -85,B 0,C 180,E1 4557.261,E2 4557.261} C_VEL
LIN {X 0,Y 514.892,Z 680.77,A -85,B 0,C 180,E1 4565.189,E2 4565.189} C_VEL
LIN {X 0,Y 521.969,Z 708.764,A -85,B 0,C 180,E1 4565.858,E2 4565.858} C_VEL
LIN {X 0,Y 521.419,Z 777.597,A -85,B 0,C 180,E1 4567.261,E2 4567.261} C_VEL
LIN {X 0,Y 519.464,Z 829.42,A -85,B 0,C 180,E1 4570.013,E2 4570.013} C_VEL
LIN {X 0,Y 517.661,Z 869.732,A -85,B 0,C 180,E1 4573.829,E2 4573.829} C_VEL
LIN {X 0,Y 516.233,Z 901.735,A -85,B 0,C 180,E1 4578.984,E2 4578.984} C_VEL
LIN {X 0,Y 515.588,Z 921.045,A -85,B 0,C 180,E1 4584.934,E2 4584.934} C_VEL
LIN {X 0,Y 515.248,Z 925.836,A -85,B 0,C 180,E1 4590.844,E2 4590.844} C_VEL
LIN {X 0,Y 515.255,Z 918.254,A -85,B 0,C 180,E1 4596.341,E2 4596.341} C_VEL
LIN {X 0,Y 515.854,Z 897.567,A -85,B 0,C 180,E1 4601.884,E2 4601.884} C_VEL
LIN {X 0,Y 517.604,Z 863.026,A -85,B 0,C 180,E1 4606.976,E2 4606.976} C_VEL
LIN {X 0,Y 520.018,Z 816.839,A -85,B 0,C 180,E1 4610.834,E2 4610.834} C_VEL
LIN {X 0,Y 521.959,Z 763.135,A -85,B 0,C 180,E1 4613.201,E2 4613.201} C_VEL
LIN {X 0,Y 519.926,Z 696.519,A -85,B 0,C 180,E1 4614.405,E2 4614.405} C_VEL
LIN {X 0,Y 514.081,Z 678.81,A -85,B 0,C 180,E1 4615.08,E2 4615.08} C_VEL
LIN {X 0,Y 514.304,Z 678.81,A -85,B 0,C 180,E1 4623.084,E2 4623.084} C_VEL
LIN {X 0,Y 514.295,Z 678.81,A -85,B 0,C 180,E1 4631.599,E2 4631.599} C_VEL
LIN {X 0,Y 514.155,Z 678.81,A -85,B 0,C 180,E1 4640.606,E2 4640.606} C_VEL
LIN {X 0,Y 514.274,Z 678.81,A -85,B 0,C 180,E1 4650.517,E2 4650.517} C_VEL
LIN {X 0,Y 514.074,Z 678.81,A -85,B 0,C 180,E1 4658.416,E2 4658.416} C_VEL
LIN {X 0,Y 514.46,Z 678.81,A -85,B 0,C 180,E1 4667.216,E2 4667.216} C_VEL
LIN {X 0,Y 514.829,Z 678.81,A -85,B 0,C 180,E1 4675.772,E2 4675.772} C_VEL
LIN {X 0,Y 513.99,Z 678.81,A -85,B 0,C 180,E1 4682.537,E2 4682.537} C_VEL
LIN {X 0,Y 514.805,Z 678.81,A -85,B 0,C 180,E1 4691.045,E2 4691.045} C_VEL
LIN {X 0,Y 514.572,Z 678.81,A -85,B 0,C 180,E1 4699.824,E2 4699.824} C_VEL
LIN {X 0,Y 514.466,Z 678.81,A -85,B 0,C 180,E1 4709.521,E2 4709.521} C_VEL
LIN {X 0,Y 514.331,Z 678.81,A -85,B 0,C 180,E1 4719.373,E2 4719.373} C_VEL
LIN {X 0,Y 514.369,Z 678.81,A -85,B 0,C 180,E1 4728.793,E2 4728.793} C_VEL
LIN {X 0,Y 514.27,Z 678.81,A -85,B 0,C 180,E1 4738.909,E2 4738.909} C_VEL
LIN {X 0,Y 514.24,Z 678.81,A -85,B 0,C 180,E1 4746.522,E2 4746.522} C_VEL
LIN {X 0,Y 514.621,Z 678.81,A -85,B 0,C 180,E1 4755.484,E2 4755.484} C_VEL
LIN {X 0,Y 514.923,Z 678.81,A -85,B 0,C 180,E1 4764.08,E2 4764.08} C_VEL
LIN {X 0,Y 514.501,Z 678.81,A -85,B 0,C 180,E1 4770.845,E2 4770.845} C_VEL
LIN {X 0,Y 514.516,Z 680.301,A -85,B 0,C 180,E1 4775.554,E2 4775.554} C_VEL
LIN {X 0,Y 518.048,Z 708.04,A -85,B 0,C 180,E1 4776.94,E2 4776.94} C_VEL
LIN {X 0,Y 516.631,Z 742.789,A -85,B 0,C 180,E1 4779.961,E2 4779.961} C_VEL
LIN {X 0,Y 515.749,Z 767.014,A -85,B 0,C 180,E1 4784.213,E2 4784.213} C_VEL
LIN {X 0,Y 515.452,Z 776.165,A -85,B 0,C 180,E1 4788.007,E2 4788.007} C_VEL
LIN {X 0,Y 515.578,Z 775.168,A -85,B 0,C 180,E1 4792.627,E2 4792.627} C_VEL
LIN {X 0,Y 516.209,Z 759.43,A -85,B 0,C 180,E1 4797.424,E2 4797.424} C_VEL
LIN {X 0,Y 517.348,Z 730.593,A -85,B 0,C 180,E1 4801.279,E2 4801.279} C_VEL
LIN {X 0,Y 517.727,Z 691.724,A -85,B 0,C 180,E1 4803.846,E2 4803.846} C_VEL
LIN {X 0,Y 514.656,Z 678.81,A -85,B 0,C 180,E1 4804.621,E2 4804.621} C_VEL
LIN {X 0,Y 514.247,Z 678.81,A -85,B 0,C 180,E1 4813.907,E2 4813.907} C_VEL
LIN {X 0,Y 514.032,Z 678.81,A -85,B 0,C 180,E1 4822.756,E2 4822.756} C_VEL
LIN {X 0,Y 514.306,Z 678.81,A -85,B 0,C 180,E1 4830.866,E2 4830.866} C_VEL
LIN {X 0,Y 514.137,Z 678.81,A -85,B 0,C 180,E1 4840.158,E2 4840.158} C_VEL
LIN {X 0,Y 514.573,Z 678.81,A -85,B 0,C 180,E1 4848.949,E2 4848.949} C_VEL
LIN {X 0,Y 515.218,Z 678.81,A -85,B 0,C 180,E1 4857.767,E2 4857.767} C_VEL
LIN {X 0,Y 515.015,Z 678.81,A -85,B 0,C 180,E1 4867.622,E2 4867.622} C_VEL
LIN {X 0,Y 514.604,Z 678.81,A -85,B 0,C 180,E1 4876.582,E2 4876.582} C_VEL
LIN {X 0,Y 514.516,Z 678.81,A -85,B 0,C 180,E1 4885.896,E2 4885.896} C_VEL
LIN {X 0,Y 514.43,Z 678.81,A -85,B 0,C 180,E1 4896.134,E2 4896.134} C_VEL
LIN {X 0,Y 514.319,Z 678.81,A -85,B 0,C 180,E1 4899.973,E2 4899.973} C_VEL
LIN {X 0,Y 506.282,Z 678.81,A -85,B 0,C 180,E1 4903.873,E2 4903.873} C_VEL
LIN {X 0,Y 506.322,Z 678.81,A -85,B 0,C 180,E1 4914.236,E2 4914.236} C_VEL
LIN {X 0,Y 506.589,Z 678.81,A -85,B 0,C 180,E1 4924.255,E2 4924.255} C_VEL
LIN {X 0,Y 506.888,Z 680.793,A -85,B 0,C 180,E1 4924.869,E2 4924.869} C_VEL
LIN {X 0,Y 514.439,Z 710.558,A -85,B 0,C 180,E1 4925.597,E2 4925.597} C_VEL
LIN {X 0,Y 513.76,Z 777.884,A -85,B 0,C 180,E1 4927.017,E2 4927.017} C_VEL
LIN {X 0,Y 511.572,Z 830.494,A -85,B 0,C 180,E1 4929.91,E2 4929.91} C_VEL
LIN {X 0,Y 509.524,Z 874.226,A -85,B 0,C 180,E1 4934.23,E2 4934.23} C_VEL
LIN {X 0,Y 508.22,Z 903.686,A -85,B 0,C 180,E1 4939.244,E2 4939.244} C_VEL
LIN {X 0,Y 507.624,Z 921.045,A -85,B 0,C 180,E1 4944.854,E2 4944.854} C_VEL
LIN {X 0,Y 507.26,Z 925.836,A -85,B 0,C 180,E1 4950.857,E2 4950.857} C_VEL
LIN {X 0,Y 507.264,Z 918.253,A -85,B 0,C 180,E1 4956.441,E2 4956.441} C_VEL
LIN {X 0,Y 507.923,Z 897.566,A -85,B 0,C 180,E1 4962.072,E2 4962.072} C_VEL
LIN {X 0,Y 509.599,Z 865.867,A -85,B 0,C 180,E1 4966.798,E2 4966.798} C_VEL
LIN {X 0,Y 512.169,Z 819.175,A -85,B 0,C 180,E1 4970.901,E2 4970.901} C_VEL
LIN {X 0,Y 514.233,Z 766.995,A -85,B 0,C 180,E1 4973.363,E2 4973.363} C_VEL
LIN {X 0,Y 512.404,Z 698.541,A -85,B 0,C 180,E1 4974.674,E2 4974.674} C_VEL
LIN {X 0,Y 506.024,Z 678.81,A -85,B 0,C 180,E1 4975.473,E2 4975.473} C_VEL
LIN {X 0,Y 506.147,Z 678.81,A -85,B 0,C 180,E1 4984.453,E2 4984.453} C_VEL
LIN {X 0,Y 506.192,Z 678.81,A -85,B 0,C 180,E1 4992.729,E2 4992.729} C_VEL
LIN {X 0,Y 506.051,Z 678.81,A -85,B 0,C 180,E1 5002.061,E2 5002.061} C_VEL
LIN {X 0,Y 506.29,Z 678.81,A -85,B 0,C 180,E1 5010.355,E2 5010.355} C_VEL
LIN {X 0,Y 506.095,Z 678.81,A -85,B 0,C 180,E1 5019.825,E2 5019.825} C_VEL
LIN {X 0,Y 506.536,Z 678.81,A -85,B 0,C 180,E1 5028.768,E2 5028.768} C_VEL
LIN {X 0,Y 507.182,Z 678.81,A -85,B 0,C 180,E1 5037.426,E2 5037.426} C_VEL
LIN {X 0,Y 507.092,Z 678.81,A -85,B 0,C 180,E1 5049.472,E2 5049.472} C_VEL
LIN {X 0,Y 506.559,Z 678.81,A -85,B 0,C 180,E1 5059.322,E2 5059.322} C_VEL
LIN {X 0,Y 506.419,Z 678.81,A -85,B 0,C 180,E1 5067.871,E2 5067.871} C_VEL
LIN {X 0,Y 506.221,Z 678.81,A -85,B 0,C 180,E1 5077.919,E2 5077.919} C_VEL
LIN {X 0,Y 506.31,Z 678.81,A -85,B 0,C 180,E1 5087.594,E2 5087.594} C_VEL
LIN {X 0,Y 506.28,Z 678.81,A -85,B 0,C 180,E1 5098.362,E2 5098.362} C_VEL
LIN {X 0,Y 506.247,Z 678.81,A -85,B 0,C 180,E1 5106.129,E2 5106.129} C_VEL
LIN {X 0,Y 506.637,Z 678.81,A -85,B 0,C 180,E1 5115.25,E2 5115.25} C_VEL
LIN {X 0,Y 506.923,Z 678.81,A -85,B 0,C 180,E1 5123.986,E2 5123.986} C_VEL
LIN {X 0,Y 506.511,Z 678.81,A -85,B 0,C 180,E1 5130.858,E2 5130.858} C_VEL
LIN {X 0,Y 506.458,Z 680.379,A -85,B 0,C 180,E1 5135.237,E2 5135.237} C_VEL
LIN {X 0,Y 510.473,Z 707.561,A -85,B 0,C 180,E1 5136.615,E2 5136.615} C_VEL
LIN {X 0,Y 508.939,Z 742.489,A -85,B 0,C 180,E1 5139.608,E2 5139.608} C_VEL
LIN {X 0,Y 507.908,Z 767.018,A -85,B 0,C 180,E1 5143.815,E2 5143.815} C_VEL
LIN {X 0,Y 507.522,Z 777.651,A -85,B 0,C 180,E1 5148.298,E2 5148.298} C_VEL
LIN {X 0,Y 507.73,Z 776.009,A -85,B 0,C 180,E1 5152.865,E2 5152.865} C_VEL
LIN {X 0,Y 508.41,Z 760.609,A -85,B 0,C 180,E1 5157.559,E2 5157.559} C_VEL
LIN {X 0,Y 509.616,Z 732.581,A -85,B 0,C 180,E1 5161.407,E2 5161.407} C_VEL
LIN {X 0,Y 510.435,Z 694.746,A -85,B 0,C 180,E1 5164.01,E2 5164.01} C_VEL
LIN {X 0,Y 506.62,Z 678.81,A -85,B 0,C 180,E1 5164.854,E2 5164.854} C_VEL
LIN {X 0,Y 506.211,Z 678.81,A -85,B 0,C 180,E1 5174.789,E2 5174.789} C_VEL
LIN {X 0,Y 506.161,Z 678.81,A -85,B 0,C 180,E1 5184.222,E2 5184.222} C_VEL
LIN {X 0,Y 506.51,Z 678.81,A -85,B 0,C 180,E1 5194.251,E2 5194.251} C_VEL
LIN {X 0,Y 506.628,Z 678.81,A -85,B 0,C 180,E1 5205.251,E2 5205.251} C_VEL
LIN {X 0,Y 506.916,Z 678.81,A -85,B 0,C 180,E1 5213.987,E2 5213.987} C_VEL
LIN {X 0,Y 507.002,Z 678.81,A -85,B 0,C 180,E1 5220.859,E2 5220.859} C_VEL
LIN {X 0,Y 506.749,Z 678.81,A -85,B 0,C 180,E1 5229.483,E2 5229.483} C_VEL
LIN {X 0,Y 506.715,Z 678.81,A -85,B 0,C 180,E1 5239.372,E2 5239.372} C_VEL
LIN {X 0,Y 506.506,Z 678.81,A -85,B 0,C 180,E1 5249.631,E2 5249.631} C_VEL
LIN {X 0,Y 506.452,Z 678.81,A -85,B 0,C 180,E1 5257.903,E2 5257.903} C_VEL
LIN {X 0,Y 506.282,Z 678.81,A -85,B 0,C 180,E1 5263.873,E2 5263.873} C_VEL
LIN {X 0,Y 498.149,Z 678.81,A -85,B 0,C 180,E1 5267.827,E2 5267.827} C_VEL
LIN {X 0,Y 498.191,Z 678.81,A -85,B 0,C 180,E1 5277.787,E2 5277.787} C_VEL
LIN {X 0,Y 498.835,Z 680.732,A -85,B 0,C 180,E1 5284.534,E2 5284.534} C_VEL
LIN {X 0,Y 506.925,Z 713.17,A -85,B 0,C 180,E1 5285.34,E2 5285.34} C_VEL
LIN {X 0,Y 506.086,Z 778.142,A -85,B 0,C 180,E1 5286.765,E2 5286.765} C_VEL
LIN {X 0,Y 503.746,Z 830.593,A -85,B 0,C 180,E1 5289.73,E2 5289.73} C_VEL
LIN {X 0,Y 501.54,Z 874.478,A -85,B 0,C 180,E1 5294.198,E2 5294.198} C_VEL
LIN {X 0,Y 500.123,Z 905.256,A -85,B 0,C 180,E1 5299.51,E2 5299.51} C_VEL
LIN {X 0,Y 499.317,Z 922.59,A -85,B 0,C 180,E1 5305.642,E2 5305.642} C_VEL
LIN {X 0,Y 499.256,Z 925.836,A -85,B 0,C 180,E1 5310.871,E2 5310.871} C_VEL
LIN {X 0,Y 499.251,Z 918.253,A -85,B 0,C 180,E1 5316.545,E2 5316.545} C_VEL
LIN {X 0,Y 499.949,Z 897.938,A -85,B 0,C 180,E1 5322.045,E2 5322.045} C_VEL
LIN {X 0,Y 501.773,Z 862.999,A -85,B 0,C 180,E1 5327.234,E2 5327.234} C_VEL
LIN {X 0,Y 504.479,Z 816.188,A -85,B 0,C 180,E1 5331.312,E2 5331.312} C_VEL
LIN {X 0,Y 506.731,Z 764.094,A -85,B 0,C 180,E1 5333.73,E2 5333.73} C_VEL
LIN {X 0,Y 505.038,Z 700.689,A -85,B 0,C 180,E1 5334.943,E2 5334.943} C_VEL
LIN {X 0,Y 498.038,Z 678.81,A -85,B 0,C 180,E1 5335.797,E2 5335.797} C_VEL
LIN {X 0,Y 498.18,Z 678.81,A -85,B 0,C 180,E1 5344.301,E2 5344.301} C_VEL
LIN {X 0,Y 498.166,Z 678.81,A -85,B 0,C 180,E1 5354.279,E2 5354.279} C_VEL
LIN {X 0,Y 498.146,Z 678.81,A -85,B 0,C 180,E1 5363.832,E2 5363.832} C_VEL
LIN {X 0,Y 498.441,Z 678.81,A -85,B 0,C 180,E1 5373.916,E2 5373.916} C_VEL
LIN {X 0,Y 498.623,Z 678.81,A -85,B 0,C 180,E1 5385.005,E2 5385.005} C_VEL
LIN {X 0,Y 498.909,Z 678.81,A -85,B 0,C 180,E1 5393.887,E2 5393.887} C_VEL
LIN {X 0,Y 498.465,Z 678.81,A -85,B 0,C 180,E1 5400.87,E2 5400.87} C_VEL
LIN {X 0,Y 499.044,Z 678.81,A -85,B 0,C 180,E1 5409.627,E2 5409.627} C_VEL
LIN {X 0,Y 498.625,Z 678.81,A -85,B 0,C 180,E1 5418.636,E2 5418.636} C_VEL
LIN {X 0,Y 498.401,Z 678.81,A -85,B 0,C 180,E1 5428.161,E2 5428.161} C_VEL
LIN {X 0,Y 498.155,Z 678.81,A -85,B 0,C 180,E1 5438.646,E2 5438.646} C_VEL
LIN {X 0,Y 498.204,Z 678.81,A -85,B 0,C 180,E1 5448.27,E2 5448.27} C_VEL
LIN {X 0,Y 498.212,Z 678.81,A -85,B 0,C 180,E1 5457.789,E2 5457.789} C_VEL
LIN {X 0,Y 498.278,Z 678.81,A -85,B 0,C 180,E1 5465.723,E2 5465.723} C_VEL
LIN {X 0,Y 498.619,Z 678.81,A -85,B 0,C 180,E1 5475.007,E2 5475.007} C_VEL
LIN {X 0,Y 498.921,Z 678.81,A -85,B 0,C 180,E1 5483.889,E2 5483.889} C_VEL
LIN {X 0,Y 498.499,Z 678.81,A -85,B 0,C 180,E1 5490.872,E2 5490.872} C_VEL
LIN {X 0,Y 498.424,Z 680.587,A -85,B 0,C 180,E1 5494.912,E2 5494.912} C_VEL
LIN {X 0,Y 502.842,Z 708.959,A -85,B 0,C 180,E1 5496.39,E2 5496.39} C_VEL
LIN {X 0,Y 501.135,Z 744.901,A -85,B 0,C 180,E1 5499.587,E2 5499.587} C_VEL
LIN {X 0,Y 500.088,Z 767.722,A -85,B 0,C 180,E1 5503.595,E2 5503.595} C_VEL
LIN {X 0,Y 499.614,Z 779.117,A -85,B 0,C 180,E1 5508.598,E2 5508.598} C_VEL
LIN {X 0,Y 499.986,Z 775.654,A -85,B 0,C 180,E1 5513.713,E2 5513.713} C_VEL
LIN {X 0,Y 500.866,Z 757.963,A -85,B 0,C 180,E1 5518.417,E2 5518.417} C_VEL
LIN {X 0,Y 502.234,Z 728.889,A -85,B 0,C 180,E1 5522.077,E2 5522.077} C_VEL
LIN {X 0,Y 501.71,Z 690.765,A -85,B 0,C 180,E1 5524.55,E2 5524.55} C_VEL
LIN {X 0,Y 498.559,Z 678.81,A -85,B 0,C 180,E1 5525.193,E2 5525.193} C_VEL
LIN {X 0,Y 498.2,Z 678.81,A -85,B 0,C 180,E1 5535.711,E2 5535.711} C_VEL
LIN {X 0,Y 498.269,Z 678.81,A -85,B 0,C 180,E1 5545.706,E2 5545.706} C_VEL
LIN {X 0,Y 498.34,Z 678.81,A -85,B 0,C 180,E1 5555.726,E2 5555.726} C_VEL
LIN {X 0,Y 498.613,Z 678.81,A -85,B 0,C 180,E1 5565.008,E2 5565.008} C_VEL
LIN {X 0,Y 498.915,Z 678.81,A -85,B 0,C 180,E1 5573.89,E2 5573.89} C_VEL
LIN {X 0,Y 498.996,Z 678.81,A -85,B 0,C 180,E1 5580.873,E2 5580.873} C_VEL
LIN {X 0,Y 498.75,Z 678.81,A -85,B 0,C 180,E1 5589.636,E2 5589.636} C_VEL
LIN {X 0,Y 498.666,Z 678.81,A -85,B 0,C 180,E1 5598.638,E2 5598.638} C_VEL
LIN {X 0,Y 498.526,Z 678.81,A -85,B 0,C 180,E1 5608.157,E2 5608.157} C_VEL
LIN {X 0,Y 498.33,Z 678.81,A -85,B 0,C 180,E1 5618.634,E2 5618.634} C_VEL
LIN {X 0,Y 498.149,Z 678.81,A -85,B 0,C 180,E1 5627.827,E2 5627.827} C_VEL
LIN {X 0,Y 490.177,Z 678.81,A -85,B 0,C 180,E1 5631.849,E2 5631.849} C_VEL
LIN {X 0,Y 490.563,Z 678.81,A -85,B 0,C 180,E1 5641.851,E2 5641.851} C_VEL
LIN {X 0,Y 490.826,Z 680.687,A -85,B 0,C 180,E1 5644.186,E2 5644.186} C_VEL
LIN {X 0,Y 499.37,Z 712.77,A -85,B 0,C 180,E1 5645.028,E2 5645.028} C_VEL
LIN {X 0,Y 498.49,Z 776.952,A -85,B 0,C 180,E1 5646.449,E2 5646.449} C_VEL
LIN {X 0,Y 496.028,Z 828.841,A -85,B 0,C 180,E1 5649.401,E2 5649.401} C_VEL
LIN {X 0,Y 493.683,Z 873.053,A -85,B 0,C 180,E1 5653.939,E2 5653.939} C_VEL
LIN {X 0,Y 492.195,Z 903.99,A -85,B 0,C 180,E1 5659.339,E2 5659.339} C_VEL
LIN {X 0,Y 491.376,Z 922.075,A -85,B 0,C 180,E1 5665.572,E2 5665.572} C_VEL
LIN {X 0,Y 491.286,Z 925.522,A -85,B 0,C 180,E1 5670.885,E2 5670.885} C_VEL
LIN {X 0,Y 491.269,Z 917.443,A -85,B 0,C 180,E1 5676.652,E2 5676.652} C_VEL
LIN {X 0,Y 491.956,Z 896.659,A -85,B 0,C 180,E1 5682.244,E2 5682.244} C_VEL
LIN {X 0,Y 493.871,Z 862.189,A -85,B 0,C 180,E1 5687.446,E2 5687.446} C_VEL
LIN {X 0,Y 496.735,Z 815.45,A -85,B 0,C 180,E1 5691.588,E2 5691.588} C_VEL
LIN {X 0,Y 499.165,Z 762.918,A -85,B 0,C 180,E1 5694.052,E2 5694.052} C_VEL
LIN {X 0,Y 497.541,Z 702.671,A -85,B 0,C 180,E1 5695.227,E2 5695.227} C_VEL
LIN {X 0,Y 490.013,Z 678.81,A -85,B 0,C 180,E1 5696.082,E2 5696.082} C_VEL
LIN {X 0,Y 490.131,Z 678.81,A -85,B 0,C 180,E1 5704.945,E2 5704.945} C_VEL
LIN {X 0,Y 490.158,Z 678.81,A -85,B 0,C 180,E1 5714.155,E2 5714.155} C_VEL
LIN {X 0,Y 490.003,Z 678.81,A -85,B 0,C 180,E1 5722.844,E2 5722.844} C_VEL
LIN {X 0,Y 490.351,Z 678.81,A -85,B 0,C 180,E1 5731.887,E2 5731.887} C_VEL
LIN {X 0,Y 490.594,Z 678.81,A -85,B 0,C 180,E1 5742.908,E2 5742.908} C_VEL
LIN {X 0,Y 491.05,Z 678.81,A -85,B 0,C 180,E1 5752.004,E2 5752.004} C_VEL
LIN {X 0,Y 490.451,Z 678.81,A -85,B 0,C 180,E1 5760.885,E2 5760.885} C_VEL
LIN {X 0,Y 490.996,Z 678.81,A -85,B 0,C 180,E1 5769.786,E2 5769.786} C_VEL
LIN {X 0,Y 490.556,Z 678.81,A -85,B 0,C 180,E1 5779.348,E2 5779.348} C_VEL
LIN {X 0,Y 490.396,Z 678.81,A -85,B 0,C 180,E1 5788.662,E2 5788.662} C_VEL
LIN {X 0,Y 490.147,Z 678.81,A -85,B 0,C 180,E1 5799.398,E2 5799.398} C_VEL
LIN {X 0,Y 490.086,Z 678.81,A -85,B 0,C 180,E1 5809.345,E2 5809.345} C_VEL
LIN {X 0,Y 490.155,Z 678.81,A -85,B 0,C 180,E1 5819.28,E2 5819.28} C_VEL
LIN {X 0,Y 490.017,Z 678.81,A -85,B 0,C 180,E1 5829.136,E2 5829.136} C_VEL
LIN {X 0,Y 490.499,Z 678.81,A -85,B 0,C 180,E1 5838.399,E2 5838.399} C_VEL
LIN {X 0,Y 491.178,Z 678.81,A -85,B 0,C 180,E1 5847.344,E2 5847.344} C_VEL
LIN {X 0,Y 490.23,Z 680.137,A -85,B 0,C 180,E1 5854.55,E2 5854.55} C_VEL
LIN {X 0,Y 495.309,Z 708.477,A -85,B 0,C 180,E1 5856.046,E2 5856.046} C_VEL
LIN {X 0,Y 493.523,Z 743.391,A -85,B 0,C 180,E1 5859.067,E2 5859.067} C_VEL
LIN {X 0,Y 492.266,Z 768.431,A -85,B 0,C 180,E1 5863.368,E2 5863.368} C_VEL
LIN {X 0,Y 491.772,Z 779.704,A -85,B 0,C 180,E1 5867.974,E2 5867.974} C_VEL
LIN {X 0,Y 491.911,Z 778.836,A -85,B 0,C 180,E1 5872.683,E2 5872.683} C_VEL
LIN {X 0,Y 492.618,Z 764.513,A -85,B 0,C 180,E1 5877.522,E2 5877.522} C_VEL
LIN {X 0,Y 494.119,Z 737.179,A -85,B 0,C 180,E1 5881.603,E2 5881.603} C_VEL
LIN {X 0,Y 495.556,Z 699.232,A -85,B 0,C 180,E1 5884.434,E2 5884.434} C_VEL
LIN {X 0,Y 490.514,Z 678.81,A -85,B 0,C 180,E1 5885.652,E2 5885.652} C_VEL
LIN {X 0,Y 490.198,Z 678.81,A -85,B 0,C 180,E1 5895.849,E2 5895.849} C_VEL
LIN {X 0,Y 490.181,Z 678.81,A -85,B 0,C 180,E1 5905.126,E2 5905.126} C_VEL
LIN {X 0,Y 490.355,Z 678.81,A -85,B 0,C 180,E1 5915.305,E2 5915.305} C_VEL
LIN {X 0,Y 490.621,Z 678.81,A -85,B 0,C 180,E1 5924.758,E2 5924.758} C_VEL
LIN {X 0,Y 490.927,Z 678.81,A -85,B 0,C 180,E1 5933.79,E2 5933.79} C_VEL
LIN {X 0,Y 491.013,Z 678.81,A -85,B 0,C 180,E1 5940.887,E2 5940.887} C_VEL
LIN {X 0,Y 490.739,Z 678.81,A -85,B 0,C 180,E1 5949.795,E2 5949.795} C_VEL
LIN {X 0,Y 490.618,Z 678.81,A -85,B 0,C 180,E1 5959.368,E2 5959.368} C_VEL
LIN {X 0,Y 490.478,Z 678.81,A -85,B 0,C 180,E1 5968.661,E2 5968.661} C_VEL
LIN {X 0,Y 490.297,Z 678.81,A -85,B 0,C 180,E1 5977.883,E2 5977.883} C_VEL
LIN {X 0,Y 490.154,Z 678.81,A -85,B 0,C 180,E1 5987.829,E2 5987.829} C_VEL
LIN {X 0,Y 490.177,Z 678.81,A -85,B 0,C 180,E1 5991.849,E2 5991.849} C_VEL
LIN {X 0,Y 482.067,Z 678.81,A -85,B 0,C 180,E1 5995.938,E2 5995.938} C_VEL
LIN {X 0,Y 482.784,Z 680.764,A -85,B 0,C 180,E1 6003.823,E2 6003.823} C_VEL
LIN {X 0,Y 491.907,Z 715.089,A -85,B 0,C 180,E1 6004.749,E2 6004.749} C_VEL
LIN {X 0,Y 490.813,Z 778.014,A -85,B 0,C 180,E1 6006.212,E2 6006.212} C_VEL
LIN {X 0,Y 488.136,Z 829.989,A -85,B 0,C 180,E1 6009.29,E2 6009.29} C_VEL
LIN {X 0,Y 485.717,Z 873.298,A -85,B 0,C 180,E1 6013.902,E2 6013.902} C_VEL
LIN {X 0,Y 484.13,Z 904.549,A -85,B 0,C 180,E1 6019.616,E2 6019.616} C_VEL
LIN {X 0,Y 483.473,Z 920.89,A -85,B 0,C 180,E1 6025.499,E2 6025.499} C_VEL
LIN {X 0,Y 483.364,Z 924.358,A -85,B 0,C 180,E1 6030.899,E2 6030.899} C_VEL
LIN {X 0,Y 483.321,Z 916.25,A -85,B 0,C 180,E1 6036.762,E2 6036.762} C_VEL
LIN {X 0,Y 483.997,Z 895.382,A -85,B 0,C 180,E1 6042.448,E2 6042.448} C_VEL
LIN {X 0,Y 485.972,Z 861.85,A -85,B 0,C 180,E1 6047.609,E2 6047.609} C_VEL
LIN {X 0,Y 488.946,Z 816.103,A -85,B 0,C 180,E1 6051.781,E2 6051.781} C_VEL
LIN {X 0,Y 491.563,Z 763.987,A -85,B 0,C 180,E1 6054.317,E2 6054.317} C_VEL
LIN {X 0,Y 489.897,Z 704.311,A -85,B 0,C 180,E1 6055.533,E2 6055.533} C_VEL
LIN {X 0,Y 482.017,Z 678.81,A -85,B 0,C 180,E1 6056.372,E2 6056.372} C_VEL
LIN {X 0,Y 482.043,Z 678.81,A -85,B 0,C 180,E1 6065.62,E2 6065.62} C_VEL
LIN {X 0,Y 482.142,Z 678.81,A -85,B 0,C 180,E1 6075.088,E2 6075.088} C_VEL
LIN {X 0,Y 482.061,Z 678.81,A -85,B 0,C 180,E1 6084.377,E2 6084.377} C_VEL
LIN {X 0,Y 482.314,Z 678.81,A -85,B 0,C 180,E1 6093.73,E2 6093.73} C_VEL
LIN {X 0,Y 482.595,Z 678.81,A -85,B 0,C 180,E1 6104.494,E2 6104.494} C_VEL
LIN {X 0,Y 482.916,Z 678.81,A -85,B 0,C 180,E1 6113.683,E2 6113.683} C_VEL
LIN {X 0,Y 482.438,Z 678.81,A -85,B 0,C 180,E1 6120.899,E2 6120.899} C_VEL
LIN {X 0,Y 482.973,Z 678.81,A -85,B 0,C 180,E1 6129.95,E2 6129.95} C_VEL
LIN {X 0,Y 482.573,Z 678.81,A -85,B 0,C 180,E1 6139.28,E2 6139.28} C_VEL
LIN {X 0,Y 482.324,Z 678.81,A -85,B 0,C 180,E1 6149.188,E2 6149.188} C_VEL
LIN {X 0,Y 482.148,Z 678.81,A -85,B 0,C 180,E1 6160.183,E2 6160.183} C_VEL
LIN {X 0,Y 481.998,Z 678.81,A -85,B 0,C 180,E1 6170.478,E2 6170.478} C_VEL
LIN {X 0,Y 482.151,Z 678.81,A -85,B 0,C 180,E1 6180.8,E2 6180.8} C_VEL
LIN {X 0,Y 482.195,Z 678.81,A -85,B 0,C 180,E1 6190.704,E2 6190.704} C_VEL
LIN {X 0,Y 482.826,Z 678.81,A -85,B 0,C 180,E1 6200.045,E2 6200.045} C_VEL
LIN {X 0,Y 483.367,Z 678.81,A -85,B 0,C 180,E1 6209.101,E2 6209.101} C_VEL
LIN {X 0,Y 482.347,Z 680.83,A -85,B 0,C 180,E1 6214.229,E2 6214.229} C_VEL
LIN {X 0,Y 487.719,Z 709.865,A -85,B 0,C 180,E1 6215.804,E2 6215.804} C_VEL
LIN {X 0,Y 485.736,Z 745.476,A -85,B 0,C 180,E1 6218.987,E2 6218.987} C_VEL
LIN {X 0,Y 484.455,Z 769.109,A -85,B 0,C 180,E1 6223.127,E2 6223.127} C_VEL
LIN {X 0,Y 483.96,Z 780.092,A -85,B 0,C 180,E1 6227.331,E2 6227.331} C_VEL
LIN {X 0,Y 484.091,Z 779.469,A -85,B 0,C 180,E1 6233.07,E2 6233.07} C_VEL
LIN {X 0,Y 484.978,Z 764.141,A -85,B 0,C 180,E1 6237.993,E2 6237.993} C_VEL
LIN {X 0,Y 486.593,Z 736.092,A -85,B 0,C 180,E1 6242.066,E2 6242.066} C_VEL
LIN {X 0,Y 487.434,Z 697.429,A -85,B 0,C 180,E1 6244.893,E2 6244.893} C_VEL
LIN {X 0,Y 482.502,Z 678.81,A -85,B 0,C 180,E1 6245.872,E2 6245.872} C_VEL
LIN {X 0,Y 482.124,Z 678.81,A -85,B 0,C 180,E1 6255.09,E2 6255.09} C_VEL
LIN {X 0,Y 482.028,Z 678.81,A -85,B 0,C 180,E1 6264.379,E2 6264.379} C_VEL
LIN {X 0,Y 482.343,Z 678.81,A -85,B 0,C 180,E1 6273.723,E2 6273.723} C_VEL
LIN {X 0,Y 482.585,Z 678.81,A -85,B 0,C 180,E1 6284.498,E2 6284.498} C_VEL
LIN {X 0,Y 482.922,Z 678.81,A -85,B 0,C 180,E1 6293.687,E2 6293.687} C_VEL
LIN {X 0,Y 483.007,Z 678.81,A -85,B 0,C 180,E1 6300.902,E2 6300.902} C_VEL
LIN {X 0,Y 482.742,Z 678.81,A -85,B 0,C 180,E1 6309.959,E2 6309.959} C_VEL
LIN {X 0,Y 482.632,Z 678.81,A -85,B 0,C 180,E1 6319.281,E2 6319.281} C_VEL
LIN {X 0,Y 482.378,Z 678.81,A -85,B 0,C 180,E1 6329.188,E2 6329.188} C_VEL
LIN {X 0,Y 482.284,Z 678.81,A -85,B 0,C 180,E1 6339.564,E2 6339.564} C_VEL
LIN {X 0,Y 482.177,Z 678.81,A -85,B 0,C 180,E1 6349.82,E2 6349.82} C_VEL
LIN {X 0,Y 482.067,Z 678.81,A -85,B 0,C 180,E1 6355.938,E2 6355.938} C_VEL
LIN {X 0,Y 474.299,Z 678.81,A -85,B 0,C 180,E1 6360.091,E2 6360.091} C_VEL
LIN {X 0,Y 474.754,Z 680.817,A -85,B 0,C 180,E1 6363.447,E2 6363.447} C_VEL
LIN {X 0,Y 484.456,Z 717.152,A -85,B 0,C 180,E1 6364.452,E2 6364.452} C_VEL
LIN {X 0,Y 483.18,Z 778.238,A -85,B 0,C 180,E1 6365.931,E2 6365.931} C_VEL
LIN {X 0,Y 480.321,Z 830.063,A -85,B 0,C 180,E1 6369.09,E2 6369.09} C_VEL
LIN {X 0,Y 477.819,Z 871.856,A -85,B 0,C 180,E1 6373.628,E2 6373.628} C_VEL
LIN {X 0,Y 476.209,Z 903.277,A -85,B 0,C 180,E1 6379.442,E2 6379.442} C_VEL
LIN {X 0,Y 475.587,Z 919.706,A -85,B 0,C 180,E1 6385.424,E2 6385.424} C_VEL
LIN {X 0,Y 475.442,Z 923.192,A -85,B 0,C 180,E1 6390.914,E2 6390.914} C_VEL
LIN {X 0,Y 475.37,Z 915.056,A -85,B 0,C 180,E1 6396.875,E2 6396.875} C_VEL
LIN {X 0,Y 476.083,Z 894.24,A -85,B 0,C 180,E1 6402.632,E2 6402.632} C_VEL
LIN {X 0,Y 478.071,Z 860.34,A -85,B 0,C 180,E1 6407.916,E2 6407.916} C_VEL
LIN {X 0,Y 481.256,Z 814.787,A -85,B 0,C 180,E1 6412.111,E2 6412.111} C_VEL
LIN {X 0,Y 484.051,Z 762.584,A -85,B 0,C 180,E1 6414.667,E2 6414.667} C_VEL
LIN {X 0,Y 482.546,Z 706.549,A -85,B 0,C 180,E1 6415.82,E2 6415.82} C_VEL
LIN {X 0,Y 474.004,Z 678.81,A -85,B 0,C 180,E1 6416.738,E2 6416.738} C_VEL
LIN {X 0,Y 474.03,Z 678.81,A -85,B 0,C 180,E1 6426.317,E2 6426.317} C_VEL
LIN {X 0,Y 474.094,Z 678.81,A -85,B 0,C 180,E1 6436.506,E2 6436.506} C_VEL
LIN {X 0,Y 474.111,Z 678.81,A -85,B 0,C 180,E1 6445.93,E2 6445.93} C_VEL
LIN {X 0,Y 474.156,Z 678.81,A -85,B 0,C 180,E1 6455.804,E2 6455.804} C_VEL
LIN {X 0,Y 474.48,Z 678.81,A -85,B 0,C 180,E1 6466.118,E2 6466.118} C_VEL
LIN {X 0,Y 474.837,Z 678.81,A -85,B 0,C 180,E1 6475.415,E2 6475.415} C_VEL
LIN {X 0,Y 473.985,Z 678.81,A -85,B 0,C 180,E1 6482.751,E2 6482.751} C_VEL
LIN {X 0,Y 474.929,Z 678.81,A -85,B 0,C 180,E1 6490.121,E2 6490.121} C_VEL
LIN {X 0,Y 474.553,Z 678.81,A -85,B 0,C 180,E1 6499.619,E2 6499.619} C_VEL
LIN {X 0,Y 474.32,Z 678.81,A -85,B 0,C 180,E1 6509.729,E2 6509.729} C_VEL
LIN {X 0,Y 474.066,Z 678.81,A -85,B 0,C 180,E1 6518.625,E2 6518.625} C_VEL
LIN {X 0,Y 474.011,Z 678.81,A -85,B 0,C 180,E1 6528.981,E2 6528.981} C_VEL
LIN {X 0,Y 474.093,Z 678.81,A -85,B 0,C 180,E1 6538.119,E2 6538.119} C_VEL
LIN {X 0,Y 474.067,Z 678.81,A -85,B 0,C 180,E1 6546.413,E2 6546.413} C_VEL
LIN {X 0,Y 474.472,Z 678.81,A -85,B 0,C 180,E1 6556.121,E2 6556.121} C_VEL
LIN {X 0,Y 474.85,Z 678.81,A -85,B 0,C 180,E1 6565.417,E2 6565.417} C_VEL
LIN {X 0,Y 474.061,Z 678.81,A -85,B 0,C 180,E1 6572.752,E2 6572.752} C_VEL
LIN {X 0,Y 474.329,Z 680.873,A -85,B 0,C 180,E1 6573.87,E2 6573.87} C_VEL
LIN {X 0,Y 480.09,Z 711.633,A -85,B 0,C 180,E1 6575.581,E2 6575.581} C_VEL
LIN {X 0,Y 477.987,Z 747.027,A -85,B 0,C 180,E1 6578.844,E2 6578.844} C_VEL
LIN {X 0,Y 476.563,Z 771.301,A -85,B 0,C 180,E1 6583.284,E2 6583.284} C_VEL
LIN {X 0,Y 476.01,Z 781.71,A -85,B 0,C 180,E1 6587.63,E2 6587.63} C_VEL
LIN {X 0,Y 476.129,Z 781.288,A -85,B 0,C 180,E1 6592.709,E2 6592.709} C_VEL
LIN {X 0,Y 477.032,Z 766.601,A -85,B 0,C 180,E1 6597.877,E2 6597.877} C_VEL
LIN {X 0,Y 478.821,Z 739.234,A -85,B 0,C 180,E1 6602.09,E2 6602.09} C_VEL
LIN {X 0,Y 480.369,Z 701.479,A -85,B 0,C 180,E1 6605.025,E2 6605.025} C_VEL
LIN {X 0,Y 474.442,Z 678.81,A -85,B 0,C 180,E1 6606.281,E2 6606.281} C_VEL
LIN {X 0,Y 474.069,Z 678.81,A -85,B 0,C 180,E1 6616.509,E2 6616.509} C_VEL
LIN {X 0,Y 474.09,Z 678.81,A -85,B 0,C 180,E1 6625.933,E2 6625.933} C_VEL
LIN {X 0,Y 474.154,Z 678.81,A -85,B 0,C 180,E1 6635.805,E2 6635.805} C_VEL
LIN {X 0,Y 474.466,Z 678.81,A -85,B 0,C 180,E1 6646.122,E2 6646.122} C_VEL
LIN {X 0,Y 474.842,Z 678.81,A -85,B 0,C 180,E1 6655.419,E2 6655.419} C_VEL
LIN {X 0,Y 474.818,Z 678.81,A -85,B 0,C 180,E1 6662.75,E2 6662.75} C_VEL
LIN {X 0,Y 474.819,Z 678.81,A -85,B 0,C 180,E1 6671.993,E2 6671.993} C_VEL
LIN {X 0,Y 474.559,Z 678.81,A -85,B 0,C 180,E1 6681.58,E2 6681.58} C_VEL
LIN {X 0,Y 474.208,Z 678.81,A -85,B 0,C 180,E1 6692,E2 6692} C_VEL
LIN {X 0,Y 474.173,Z 678.81,A -85,B 0,C 180,E1 6701.228,E2 6701.228} C_VEL
LIN {X 0,Y 474.166,Z 678.81,A -85,B 0,C 180,E1 6711.646,E2 6711.646} C_VEL
LIN {X 0,Y 474.299,Z 678.81,A -85,B 0,C 180,E1 6720.091,E2 6720.091} C_VEL
LIN {X 0,Y 466.464,Z 678.81,A -85,B 0,C 180,E1 6722.854,E2 6722.854} C_VEL
LIN {X 0,Y 476.997,Z 719.076,A -85,B 0,C 180,E1 6724.143,E2 6724.143} C_VEL
LIN {X 0,Y 475.581,Z 778.357,A -85,B 0,C 180,E1 6725.635,E2 6725.635} C_VEL
LIN {X 0,Y 472.588,Z 828.804,A -85,B 0,C 180,E1 6728.771,E2 6728.771} C_VEL
LIN {X 0,Y 469.824,Z 872.218,A -85,B 0,C 180,E1 6733.6,E2 6733.6} C_VEL
LIN {X 0,Y 468.123,Z 903.827,A -85,B 0,C 180,E1 6739.729,E2 6739.729} C_VEL
LIN {X 0,Y 467.681,Z 918.518,A -85,B 0,C 180,E1 6745.347,E2 6745.347} C_VEL
LIN {X 0,Y 467.52,Z 922.026,A -85,B 0,C 180,E1 6750.93,E2 6750.93} C_VEL
LIN {X 0,Y 467.471,Z 914.918,A -85,B 0,C 180,E1 6756.524,E2 6756.524} C_VEL
LIN {X 0,Y 468.084,Z 894.294,A -85,B 0,C 180,E1 6762.575,E2 6762.575} C_VEL
LIN {X 0,Y 470.078,Z 861.821,A -85,B 0,C 180,E1 6767.86,E2 6767.86} C_VEL
LIN {X 0,Y 473.41,Z 816.267,A -85,B 0,C 180,E1 6772.25,E2 6772.25} C_VEL
LIN {X 0,Y 476.389,Z 764.32,A -85,B 0,C 180,E1 6774.916,E2 6774.916} C_VEL
LIN {X 0,Y 475.067,Z 708.213,A -85,B 0,C 180,E1 6776.13,E2 6776.13} C_VEL
LIN {X 0,Y 466.019,Z 678.81,A -85,B 0,C 180,E1 6777.292,E2 6777.292} C_VEL
LIN {X 0,Y 466.019,Z 678.81,A -85,B 0,C 180,E1 6787.07,E2 6787.07} C_VEL
LIN {X 0,Y 466.025,Z 678.81,A -85,B 0,C 180,E1 6797.112,E2 6797.112} C_VEL
LIN {X 0,Y 466.101,Z 678.81,A -85,B 0,C 180,E1 6807.502,E2 6807.502} C_VEL
LIN {X 0,Y 466.149,Z 678.81,A -85,B 0,C 180,E1 6815.984,E2 6815.984} C_VEL
LIN {X 0,Y 466.464,Z 678.81,A -85,B 0,C 180,E1 6825.875,E2 6825.875} C_VEL
LIN {X 0,Y 466.831,Z 678.81,A -85,B 0,C 180,E1 6835.336,E2 6835.336} C_VEL
LIN {X 0,Y 465.981,Z 678.81,A -85,B 0,C 180,E1 6842.798,E2 6842.798} C_VEL
LIN {X 0,Y 466.907,Z 678.81,A -85,B 0,C 180,E1 6850.296,E2 6850.296} C_VEL
LIN {X 0,Y 466.51,Z 678.81,A -85,B 0,C 180,E1 6859.971,E2 6859.971} C_VEL
LIN {X 0,Y 466.219,Z 678.81,A -85,B 0,C 180,E1 6870.393,E2 6870.393} C_VEL
LIN {X 0,Y 465.965,Z 678.81,A -85,B 0,C 180,E1 6880.063,E2 6880.063} C_VEL
LIN {X 0,Y 465.892,Z 678.81,A -85,B 0,C 180,E1 6889.949,E2 6889.949} C_VEL
LIN {X 0,Y 466.073,Z 678.81,A -85,B 0,C 180,E1 6899.69,E2 6899.69} C_VEL
LIN {X 0,Y 466.051,Z 678.81,A -85,B 0,C 180,E1 6910.007,E2 6910.007} C_VEL
LIN {X 0,Y 466.713,Z 678.81,A -85,B 0,C 180,E1 6919.698,E2 6919.698} C_VEL
LIN {X 0,Y 467.359,Z 678.81,A -85,B 0,C 180,E1 6929.07,E2 6929.07} C_VEL
LIN {X 0,Y 466.089,Z 679.475,A -85,B 0,C 180,E1 6933.442,E2 6933.442} C_VEL
LIN {X 0,Y 472.515,Z 712.159,A -85,B 0,C 180,E1 6935.274,E2 6935.274} C_VEL
LIN {X 0,Y 470.307,Z 747.422,A -85,B 0,C 180,E1 6938.542,E2 6938.542} C_VEL
LIN {X 0,Y 468.754,Z 771.686,A -85,B 0,C 180,E1 6942.957,E2 6942.957} C_VEL
LIN {X 0,Y 468.053,Z 783.246,A -85,B 0,C 180,E1 6947.94,E2 6947.94} C_VEL
LIN {X 0,Y 468.429,Z 780.628,A -85,B 0,C 180,E1 6953.888,E2 6953.888} C_VEL
LIN {X 0,Y 469.611,Z 764.611,A -85,B 0,C 180,E1 6958.708,E2 6958.708} C_VEL
LIN {X 0,Y 471.501,Z 736.336,A -85,B 0,C 180,E1 6962.766,E2 6962.766} C_VEL
LIN {X 0,Y 471.491,Z 697.287,A -85,B 0,C 180,E1 6965.672,E2 6965.672} C_VEL
LIN {X 0,Y 466.355,Z 678.81,A -85,B 0,C 180,E1 6966.755,E2 6966.755} C_VEL
LIN {X 0,Y 465.991,Z 678.81,A -85,B 0,C 180,E1 6977.116,E2 6977.116} C_VEL
LIN {X 0,Y 466.088,Z 678.81,A -85,B 0,C 180,E1 6987.505,E2 6987.505} C_VEL
LIN {X 0,Y 466.146,Z 678.81,A -85,B 0,C 180,E1 6995.988,E2 6995.988} C_VEL
LIN {X 0,Y 466.45,Z 678.81,A -85,B 0,C 180,E1 7005.878,E2 7005.878} C_VEL
LIN {X 0,Y 466.836,Z 678.81,A -85,B 0,C 180,E1 7015.34,E2 7015.34} C_VEL
LIN {X 0,Y 466.82,Z 678.81,A -85,B 0,C 180,E1 7022.797,E2 7022.797} C_VEL
LIN {X 0,Y 466.823,Z 678.81,A -85,B 0,C 180,E1 7032.201,E2 7032.201} C_VEL
LIN {X 0,Y 466.497,Z 678.81,A -85,B 0,C 180,E1 7042.009,E2 7042.009} C_VEL
LIN {X 0,Y 466.164,Z 678.81,A -85,B 0,C 180,E1 7052.493,E2 7052.493} C_VEL
LIN {X 0,Y 466.09,Z 678.81,A -85,B 0,C 180,E1 7062.897,E2 7062.897} C_VEL
LIN {X 0,Y 466.096,Z 678.81,A -85,B 0,C 180,E1 7072.963,E2 7072.963} C_VEL
LIN {X 0,Y 466.464,Z 678.81,A -85,B 0,C 180,E1 7082.854,E2 7082.854} C_VEL
LIN {X 0,Y 471.142,Z 689.958,A -85,B 0,C 180,E1 7083.417,E2 7083.417} C_VEL
LIN {X 0,Y 469.203,Z 713.587,A -85,B 0,C 180,E1 7083.692,E2 7083.692} C_VEL
LIN {X 0,Y 468.17,Z 775.198,A -85,B 0,C 180,E1 7085.194,E2 7085.194} C_VEL
LIN {X 0,Y 464.964,Z 826.166,A -85,B 0,C 180,E1 7088.323,E2 7088.323} C_VEL
LIN {X 0,Y 461.919,Z 869.498,A -85,B 0,C 180,E1 7093.127,E2 7093.127} C_VEL
LIN {X 0,Y 460.327,Z 900.724,A -85,B 0,C 180,E1 7099.073,E2 7099.073} C_VEL
LIN {X 0,Y 459.762,Z 917.328,A -85,B 0,C 180,E1 7105.267,E2 7105.267} C_VEL
LIN {X 0,Y 459.619,Z 920.865,A -85,B 0,C 180,E1 7110.946,E2 7110.946} C_VEL
LIN {X 0,Y 459.484,Z 912.282,A -85,B 0,C 180,E1 7117.264,E2 7117.264} C_VEL
LIN {X 0,Y 460.419,Z 889.72,A -85,B 0,C 180,E1 7123.49,E2 7123.49} C_VEL
LIN {X 0,Y 462.846,Z 853.485,A -85,B 0,C 180,E1 7129.015,E2 7129.015} C_VEL
LIN {X 0,Y 466.291,Z 807.398,A -85,B 0,C 180,E1 7133.115,E2 7133.115} C_VEL
LIN {X 0,Y 469.233,Z 754.611,A -85,B 0,C 180,E1 7135.531,E2 7135.531} C_VEL
LIN {X 0,Y 467.248,Z 708.706,A -85,B 0,C 180,E1 7136.487,E2 7136.487} C_VEL
LIN {X 0,Y 458.021,Z 678.81,A -85,B 0,C 180,E1 7137.637,E2 7137.637} C_VEL
LIN {X 0,Y 457.959,Z 678.81,A -85,B 0,C 180,E1 7147.809,E2 7147.809} C_VEL
LIN {X 0,Y 457.994,Z 678.81,A -85,B 0,C 180,E1 7158.204,E2 7158.204} C_VEL
LIN {X 0,Y 458.061,Z 678.81,A -85,B 0,C 180,E1 7169.098,E2 7169.098} C_VEL
LIN {X 0,Y 458.006,Z 678.81,A -85,B 0,C 180,E1 7177.599,E2 7177.599} C_VEL
LIN {X 0,Y 458.441,Z 678.81,A -85,B 0,C 180,E1 7187.572,E2 7187.572} C_VEL
LIN {X 0,Y 459.114,Z 678.81,A -85,B 0,C 180,E1 7197.156,E2 7197.156} C_VEL
LIN {X 0,Y 458.938,Z 678.81,A -85,B 0,C 180,E1 7208.556,E2 7208.556} C_VEL
LIN {X 0,Y 458.553,Z 678.81,A -85,B 0,C 180,E1 7218.323,E2 7218.323} C_VEL
LIN {X 0,Y 458.243,Z 678.81,A -85,B 0,C 180,E1 7228.697,E2 7228.697} C_VEL
LIN {X 0,Y 457.925,Z 678.81,A -85,B 0,C 180,E1 7238.851,E2 7238.851} C_VEL
LIN {X 0,Y 457.942,Z 678.81,A -85,B 0,C 180,E1 7248.213,E2 7248.213} C_VEL
LIN {X 0,Y 458.027,Z 678.81,A -85,B 0,C 180,E1 7259.1,E2 7259.1} C_VEL
LIN {X 0,Y 457.941,Z 678.81,A -85,B 0,C 180,E1 7267.599,E2 7267.599} C_VEL
LIN {X 0,Y 458.423,Z 678.81,A -85,B 0,C 180,E1 7277.574,E2 7277.574} C_VEL
LIN {X 0,Y 459.127,Z 678.81,A -85,B 0,C 180,E1 7287.158,E2 7287.158} C_VEL
LIN {X 0,Y 458.272,Z 680.661,A -85,B 0,C 180,E1 7293.108,E2 7293.108} C_VEL
LIN {X 0,Y 464.896,Z 714.869,A -85,B 0,C 180,E1 7295.104,E2 7295.104} C_VEL
LIN {X 0,Y 462.436,Z 750.907,A -85,B 0,C 180,E1 7298.652,E2 7298.652} C_VEL
LIN {X 0,Y 460.783,Z 775.104,A -85,B 0,C 180,E1 7303.483,E2 7303.483} C_VEL
LIN {X 0,Y 460.122,Z 784.733,A -85,B 0,C 180,E1 7308.26,E2 7308.26} C_VEL
LIN {X 0,Y 460.586,Z 781.133,A -85,B 0,C 180,E1 7314.321,E2 7314.321} C_VEL
LIN {X 0,Y 461.988,Z 762.79,A -85,B 0,C 180,E1 7319.484,E2 7319.484} C_VEL
LIN {X 0,Y 464.258,Z 732.424,A -85,B 0,C 180,E1 7323.535,E2 7323.535} C_VEL
LIN {X 0,Y 463.691,Z 697.953,A -85,B 0,C 180,E1 7326.048,E2 7326.048} C_VEL
LIN {X 0,Y 458.284,Z 678.81,A -85,B 0,C 180,E1 7327.281,E2 7327.281} C_VEL
LIN {X 0,Y 457.945,Z 678.81,A -85,B 0,C 180,E1 7338.212,E2 7338.212} C_VEL
LIN {X 0,Y 458.094,Z 678.81,A -85,B 0,C 180,E1 7349.105,E2 7349.105} C_VEL
LIN {X 0,Y 457.998,Z 678.81,A -85,B 0,C 180,E1 7357.602,E2 7357.602} C_VEL
LIN {X 0,Y 458.436,Z 678.81,A -85,B 0,C 180,E1 7367.576,E2 7367.576} C_VEL
LIN {X 0,Y 459.23,Z 678.81,A -85,B 0,C 180,E1 7377.906,E2 7377.906} C_VEL
LIN {X 0,Y 458.863,Z 678.81,A -85,B 0,C 180,E1 7388.561,E2 7388.561} C_VEL
LIN {X 0,Y 458.495,Z 678.81,A -85,B 0,C 180,E1 7398.33,E2 7398.33} C_VEL
LIN {X 0,Y 458.3,Z 678.81,A -85,B 0,C 180,E1 7408.698,E2 7408.698} C_VEL
LIN {X 0,Y 458.106,Z 678.81,A -85,B 0,C 180,E1 7418.879,E2 7418.879} C_VEL
LIN {X 0,Y 458.007,Z 678.81,A -85,B 0,C 180,E1 7428.209,E2 7428.209} C_VEL
LIN {X 0,Y 458.155,Z 678.81,A -85,B 0,C 180,E1 7439.109,E2 7439.109} C_VEL
LIN {X 0,Y 458.475,Z 679.447,A -85,B 0,C 180,E1 7442.591,E2 7442.591} C_VEL
LIN {X 0,Y 469.203,Z 713.587,A -85,B 0,C 180,E1 7443.692,E2 7443.692} C_VEL
LIN {X 0,Y 467.139,Z 730.64,A -85,B 0,C 180,E1 7443.858,E2 7443.858} C_VEL
LIN {X 0,Y 461.904,Z 748.346,A -85,B 0,C 180,E1 7443.965,E2 7443.965} C_VEL
LIN {X 0,Y 458.978,Z 801.195,A -85,B 0,C 180,E1 7446.236,E2 7446.236} C_VEL
LIN {X 0,Y 455.305,Z 848.355,A -85,B 0,C 180,E1 7450.277,E2 7450.277} C_VEL
LIN {X 0,Y 452.684,Z 885.129,A -85,B 0,C 180,E1 7455.68,E2 7455.68} C_VEL
LIN {X 0,Y 451.732,Z 909.381,A -85,B 0,C 180,E1 7461.98,E2 7461.98} C_VEL
LIN {X 0,Y 451.623,Z 918.455,A -85,B 0,C 180,E1 7467.111,E2 7467.111} C_VEL
LIN {X 0,Y 451.908,Z 917.534,A -85,B 0,C 180,E1 7473.851,E2 7473.851} C_VEL
LIN {X 0,Y 452.151,Z 901.473,A -85,B 0,C 180,E1 7480.637,E2 7480.637} C_VEL
LIN {X 0,Y 453.759,Z 870.874,A -85,B 0,C 180,E1 7486.818,E2 7486.818} C_VEL
LIN {X 0,Y 457.158,Z 828.361,A -85,B 0,C 180,E1 7491.758,E2 7491.758} C_VEL
LIN {X 0,Y 460.539,Z 777.119,A -85,B 0,C 180,E1 7495.062,E2 7495.062} C_VEL
LIN {X 0,Y 461.883,Z 716.788,A -85,B 0,C 180,E1 7496.617,E2 7496.617} C_VEL
LIN {X 0,Y 450.01,Z 678.81,A -85,B 0,C 180,E1 7497.812,E2 7497.812} C_VEL
LIN {X 0,Y 449.953,Z 678.81,A -85,B 0,C 180,E1 7508.605,E2 7508.605} C_VEL
LIN {X 0,Y 449.957,Z 678.81,A -85,B 0,C 180,E1 7519.362,E2 7519.362} C_VEL
LIN {X 0,Y 450.06,Z 678.81,A -85,B 0,C 180,E1 7529.297,E2 7529.297} C_VEL
LIN {X 0,Y 449.994,Z 678.81,A -85,B 0,C 180,E1 7539.258,E2 7539.258} C_VEL
LIN {X 0,Y 450.636,Z 678.81,A -85,B 0,C 180,E1 7549.324,E2 7549.324} C_VEL
LIN {X 0,Y 451.313,Z 678.81,A -85,B 0,C 180,E1 7559.035,E2 7559.035} C_VEL
LIN {X 0,Y 450.841,Z 678.81,A -85,B 0,C 180,E1 7570.667,E2 7570.667} C_VEL
LIN {X 0,Y 450.427,Z 678.81,A -85,B 0,C 180,E1 7580.716,E2 7580.716} C_VEL
LIN {X 0,Y 450.162,Z 678.81,A -85,B 0,C 180,E1 7590.725,E2 7590.725} C_VEL
LIN {X 0,Y 449.937,Z 678.81,A -85,B 0,C 180,E1 7601.125,E2 7601.125} C_VEL
LIN {X 0,Y 449.821,Z 678.81,A -85,B 0,C 180,E1 7611.382,E2 7611.382} C_VEL
LIN {X 0,Y 449.995,Z 678.81,A -85,B 0,C 180,E1 7620.726,E2 7620.726} C_VEL
LIN {X 0,Y 450.192,Z 678.81,A -85,B 0,C 180,E1 7631.323,E2 7631.323} C_VEL
LIN {X 0,Y 450.939,Z 678.81,A -85,B 0,C 180,E1 7641.29,E2 7641.29} C_VEL
LIN {X 0,Y 451.335,Z 678.81,A -85,B 0,C 180,E1 7649.037,E2 7649.037} C_VEL
LIN {X 0,Y 450.279,Z 680.483,A -85,B 0,C 180,E1 7652.717,E2 7652.717} C_VEL
LIN {X 0,Y 457.284,Z 716.216,A -85,B 0,C 180,E1 7654.84,E2 7654.84} C_VEL
LIN {X 0,Y 454.714,Z 751.722,A -85,B 0,C 180,E1 7658.396,E2 7658.396} C_VEL
LIN {X 0,Y 452.948,Z 775.882,A -85,B 0,C 180,E1 7663.247,E2 7663.247} C_VEL
LIN {X 0,Y 452.196,Z 786.154,A -85,B 0,C 180,E1 7668.591,E2 7668.591} C_VEL
LIN {X 0,Y 452.721,Z 781.571,A -85,B 0,C 180,E1 7674.772,E2 7674.772} C_VEL
LIN {X 0,Y 454.299,Z 762.159,A -85,B 0,C 180,E1 7680.034,E2 7680.034} C_VEL
LIN {X 0,Y 456.932,Z 730.208,A -85,B 0,C 180,E1 7684.146,E2 7684.146} C_VEL
LIN {X 0,Y 455.998,Z 699.007,A -85,B 0,C 180,E1 7686.415,E2 7686.415} C_VEL
LIN {X 0,Y 450.222,Z 678.81,A -85,B 0,C 180,E1 7687.616,E2 7687.616} C_VEL
LIN {X 0,Y 449.963,Z 678.81,A -85,B 0,C 180,E1 7696.478,E2 7696.478} C_VEL
LIN {X 0,Y 449.936,Z 678.81,A -85,B 0,C 180,E1 7706.185,E2 7706.185} C_VEL
LIN {X 0,Y 450.108,Z 678.81,A -85,B 0,C 180,E1 7715.075,E2 7715.075} C_VEL
LIN {X 0,Y 450.404,Z 678.81,A -85,B 0,C 180,E1 7725.364,E2 7725.364} C_VEL
LIN {X 0,Y 450.823,Z 678.81,A -85,B 0,C 180,E1 7735.174,E2 7735.174} C_VEL
LIN {X 0,Y 450.839,Z 678.81,A -85,B 0,C 180,E1 7742.896,E2 7742.896} C_VEL
LIN {X 0,Y 450.802,Z 678.81,A -85,B 0,C 180,E1 7752.642,E2 7752.642} C_VEL
LIN {X 0,Y 450.407,Z 678.81,A -85,B 0,C 180,E1 7762.8,E2 7762.8} C_VEL
LIN {X 0,Y 450.156,Z 678.81,A -85,B 0,C 180,E1 7771.506,E2 7771.506} C_VEL
LIN {X 0,Y 450.074,Z 678.81,A -85,B 0,C 180,E1 7781.115,E2 7781.115} C_VEL
LIN {X 0,Y 450.001,Z 678.81,A -85,B 0,C 180,E1 7791.4,E2 7791.4} C_VEL
LIN {X 0,Y 450.43,Z 678.859,A -85,B 0,C 180,E1 7802.142,E2 7802.142} C_VEL
LIN {X 0,Y 462.152,Z 721.501,A -85,B 0,C 180,E1 7803.462,E2 7803.462} C_VEL
LIN {X 0,Y 461.904,Z 748.346,A -85,B 0,C 180,E1 7803.965,E2 7803.965} C_VEL
LIN {X 0,Y 452.64,Z 781.9,A -85,B 0,C 180,E1 7804.834,E2 7804.834} C_VEL
LIN {X 0,Y 448.945,Z 832.063,A -85,B 0,C 180,E1 7808.381,E2 7808.381} C_VEL
LIN {X 0,Y 445.869,Z 872.645,A -85,B 0,C 180,E1 7813.438,E2 7813.438} C_VEL
LIN {X 0,Y 444.24,Z 901.714,A -85,B 0,C 180,E1 7819.668,E2 7819.668} C_VEL
LIN {X 0,Y 443.794,Z 916.255,A -85,B 0,C 180,E1 7826.078,E2 7826.078} C_VEL
LIN {X 0,Y 443.793,Z 918.537,A -85,B 0,C 180,E1 7830.98,E2 7830.98} C_VEL
LIN {X 0,Y 443.614,Z 911.348,A -85,B 0,C 180,E1 7836.876,E2 7836.876} C_VEL
LIN {X 0,Y 444.382,Z 890.446,A -85,B 0,C 180,E1 7843.257,E2 7843.257} C_VEL
LIN {X 0,Y 446.635,Z 857.444,A -85,B 0,C 180,E1 7848.831,E2 7848.831} C_VEL
LIN {X 0,Y 450.512,Z 812.313,A -85,B 0,C 180,E1 7853.316,E2 7853.316} C_VEL
LIN {X 0,Y 453.985,Z 759.428,A -85,B 0,C 180,E1 7856.058,E2 7856.058} C_VEL
LIN {X 0,Y 452.446,Z 712.414,A -85,B 0,C 180,E1 7857.133,E2 7857.133} C_VEL
LIN {X 0,Y 441.959,Z 678.81,A -85,B 0,C 180,E1 7858.453,E2 7858.453} C_VEL
LIN {X 0,Y 441.912,Z 678.81,A -85,B 0,C 180,E1 7869.442,E2 7869.442} C_VEL
